// TwinCAT 3 PLC project Tc_PLCopen_OpcUa
// Title: Tc_PLCopen_OpcUa
// Company: Beckhoff Automation GmbH
// Author: Beckhoff Automation GmbH
// ProjectVersion: 2.0
// ProgramVersion: 3.1.4020.1
// libraries:
//   Tc2_Standard, * (Beckhoff Automation GmbH)
//   Tc2_System, * (Beckhoff Automation GmbH)
//   Tc2_Utilities, * (Beckhoff Automation GmbH)
//   Tc3_Module, * (Beckhoff Automation GmbH)
//   Tc3_PLCopen_OpcUa, * (Beckhoff Automation GmbH)
// project tree:
//   DUTs/ ST_ADSReadRes.TcDUT, ST_ADSReadWriteRes.TcDUT, ST_ReadListData.TcDUT, ST_ReadListDataArrayInt.TcDUT, TcSymbolInfo.TcDUT
//   GVLs/ GVL_Tests.TcGVL
//   BECKHOFF SPECIFIC helper library/DUTs/Database/ ST_UASQLState.TcDUT
//   BECKHOFF SPECIFIC helper library/DUTs/_Internal/Database/ ST_UAMethodCall_DBRecordInsertRes.TcDUT
//   BECKHOFF SPECIFIC helper library/DUTs/_Internal/MethodCall/ ST_ADSReadState.TcDUT, ST_DeviceInfo.TcDUT, ST_UAMethodCall_AdsReadDeviceInfoRes.TcDUT, ST_UAMethodCall_AdsReadStateRes.TcDUT
//   BECKHOFF SPECIFIC helper library/POUs/Database/ UA_MethodCall_DBRecordInsert.TcPOU
//   BECKHOFF SPECIFIC helper library/POUs/MethodCall/ UA_MethodCall_ADSReadDeviceInfoReq.TcPOU, UA_MethodCall_ADSReadReq.TcPOU, UA_MethodCall_ADSReadStateReq.TcPOU, UA_MethodCall_ADSReadWriteReq.TcPOU, UA_MethodCall_ADSWriteControlReq.TcPOU, UA_MethodCall_ADSWriteReq.TcPOU
//   POUs/ PRG_READ_List.TcPOU, PRG_READ_List_woConnectIdent.TcPOU, PRG_READ_List_ArrayInt.TcPOU, MAIN.TcPOU, PRG_ADSReadDeviceInfoReq.TcPOU, PRG_ADSReadReq.TcPOU, PRG_ADSWriteReq.TcPOU, PRG_ADSWriteControlReq.TcPOU, PRG_ADSReadWriteReq.TcPOU, PRG_ADSReadStateReq.TcPOU, PRG_READ.TcPOU, PRG_WRITE.TcPOU
//   Tests_Henning/DUTs/ U_Arrays2DimInOne.TcDUT, U_Arrays3DimInOne.TcDUT, ST_UAMethodCall_CallInOut1DimParam.TcDUT, ST_UAMethodCall_CallInOut1DimStringParam.TcDUT, ST_UAMethodCall_CallInOutParam.TcDUT, U_ArraysInOne.TcDUT, U_ScalarsInOne.TcDUT
//   Tests_Henning/GVLs/ GVL_ArrayTests2DimPLC.TcGVL, GVL_ArrayTests3DimPLC.TcGVL, GVL_ArrayTests.TcGVL, GVL_ScalarTests.TcGVL
//   Tests_Henning/POUs/ PRG_2DArrayTest.TcPOU, PRG_2DArrayTest_Read.TcPOU, PRG_2DArrayTest_ReadWritten.TcPOU, PRG_2DArrayTest_Write.TcPOU, PRG_3DArrayTest.TcPOU, PRG_3DArrayTest_Read.TcPOU, PRG_3DArrayTest_ReadWritten.TcPOU, PRG_3DArrayTest_Write.TcPOU, PRG_Connect_Encrypted.TcPOU, PRG_GetBrokenHandle.TcPOU, PRG_READ_List_Henning.TcPOU, PRG_ArrayTest.TcPOU, PRG_ArrayTest_Read.TcPOU, PRG_ArrayTest_ReadWritten.TcPOU, PRG_ArrayTest_Write.TcPOU, PRG_CallInOut1DimParam.TcPOU, PRG_CallInOut1DimStringParam.TcPOU, PRG_CallInOutMultiParam.TcPOU, PRG_ScalarTest.TcPOU, PRG_ScalarTest_Read.TcPOU, PRG_ScalarTest_ReadWritten.TcPOU, PRG_ScalarTest_Write.TcPOU
//   Test_CloudSample/DUTs/ ST_CloudSampleRes.TcDUT, ST_DBSQLError.TcDUT, ST_internalSQLError.TcDUT
//   Test_CloudSample/GVLs/ GVL_CloudSample.TcGVL
//   Test_CloudSample/POUs/ADS/ FB_CloudAdsSqlInsert.TcPOU
//   Test_CloudSample/POUs/ CloudSample.TcPOU, CloudSample_SQL.TcPOU
//   Test_CloudSample/POUs/Helper/ FB_BuildSQLInsert.TcPOU
//   / PlcTask.TcTTO
//   Test_Manz/DUTs/ ST_UAMethodCall_CallTestMethodArray.TcDUT, ST_UAMethodCall_CallTestMethodIntArray3Dim.TcDUT
//   Test_Manz/POUs/ PRG_CallTestMethodIntArray3Dim.TcPOU, PRG_CallTestMethodStringArray2Dim.TcPOU
// real-time tasks:
//   TASK PlcTask: cycle T#10ms, priority 20, ADS port 350

CONFIGURATION Tc_PLCopen_OpcUa
    RESOURCE PLC ON TwinCAT3
        TASK PlcTask(INTERVAL := T#10ms, PRIORITY := 20);
        PROGRAM MAIN WITH PlcTask : MAIN;
    END_RESOURCE
END_CONFIGURATION

// ---- DUTs/ST_ADSReadRes.TcDUT
TYPE ST_ADSReadRes :
STRUCT
	nNumberOfOutputArguments	: UDINT;
	nReserved					: ARRAY [1..4] OF BYTE; // padding
	stOutputArgInfo				: ST_UAMethodArgInfo;
	nReadData					: INT; 
END_STRUCT
END_TYPE

// ---- DUTs/ST_ADSReadWriteRes.TcDUT
TYPE ST_ADSReadWriteRes :
STRUCT
	nNumberOfOutputArguments	: UDINT;
	nReserved					: ARRAY [1..4] OF BYTE; // padding
	stOutputArgInfo				: ST_UAMethodArgInfo;
	arrAddr						: T_IPv4AddrArr	:=[ 0, 0, 0, 0];
END_STRUCT
END_TYPE

// ---- DUTs/ST_ReadListData.TcDUT
{attribute 'pack_mode' := '1'}
TYPE ST_ReadListData :
STRUCT
	stReadListReturnInfo	: ARRAY [1..gNodeIDCount] OF ST_UAReadListReturnInfo; // must be less than nMaxNodeIDsInList, nMaxNodeIDsInList = 10
	nIntVar1				: INT; 
	nIntVar2				: INT; 
	nIntVar3				: INT;
	nIntVar4				: INT;
	nIntVar5				: INT;
	nIntVar6				: INT;
	nIntVar7				: INT;
	nIntVar8				: INT;
	nIntVar9				: INT;
	nIntVar10				: INT;
END_STRUCT
END_TYPE

// ---- DUTs/ST_ReadListDataArrayInt.TcDUT
{attribute 'pack_mode' := '1'}
TYPE ST_ReadListDataArrayInt :
STRUCT
	stReadListReturnInfo	: ARRAY [1..gNodeIDCount_Array] OF ST_UAReadListReturnInfo; // must be less than nMaxNodeIDsInList, nMaxNodeIDsInList = 10
	nArrIntVar1				: ARRAY [1..10] OF INT; 
	nArrDintVar2			: ARRAY [1..2] OF DINT; 	
END_STRUCT
END_TYPE

// ---- DUTs/TcSymbolInfo.TcDUT
TYPE TcSymbolInfo :
STRUCT
	nAddress	: UDINT; 
	nLength		: UDINT; 
END_STRUCT
END_TYPE

// ---- BECKHOFF SPECIFIC helper library/DUTs/Database/ST_UASQLState.TcDUT
TYPE ST_UASQLState :
STRUCT
	sSQLState 		: STRING(5);
	nReserved		: ARRAY [1..2] OF BYTE; //padding
	nSQLErrorCode 	: DINT;
	nReturnCode		: UDINT;
END_STRUCT
END_TYPE

// ---- BECKHOFF SPECIFIC helper library/DUTs/_Internal/Database/ST_UAMethodCall_DBRecordInsertRes.TcDUT
TYPE ST_UAMethodCall_DBRecordInsertRes :
STRUCT
	nNumberOfOutputArguments	: UDINT;
	nReserved					: ARRAY [1..4] OF BYTE; // padding
	stOutputArgInfo				: ARRAY [1..1] OF ST_UAMethodArgInfo;
	stSQLStateInternal			: ST_UASQLState; 
END_STRUCT
END_TYPE

// ---- BECKHOFF SPECIFIC helper library/DUTs/_Internal/MethodCall/ST_ADSReadState.TcDUT
TYPE ST_ADSReadState :
STRUCT
	nAdsState			: DINT;			(* ADS state *)
	nDeviceState		: DINT;			(* Device state *)
END_STRUCT
END_TYPE

// ---- BECKHOFF SPECIFIC helper library/DUTs/_Internal/MethodCall/ST_DeviceInfo.TcDUT
TYPE ST_DeviceInfo :
STRUCT
	sDeviceName		: STRING(19);		(* ADS state *)
	nVersion		: SINT;				(* Device state *)
	nRevision		: SINT;
	nBuild			: INT;
END_STRUCT
END_TYPE

// ---- BECKHOFF SPECIFIC helper library/DUTs/_Internal/MethodCall/ST_UAMethodCall_AdsReadDeviceInfoRes.TcDUT
TYPE ST_UAMethodCall_AdsReadDeviceInfoRes :
STRUCT
	nNumberOfOutputArguments	: UDINT;
	nReserved					: ARRAY [1..4] OF BYTE; // padding
	stOutputArgInfo				: ARRAY [1..4] OF ST_UAMethodArgInfo;
	stDeviceInfo				: ST_DeviceInfo;
END_STRUCT
END_TYPE

// ---- BECKHOFF SPECIFIC helper library/DUTs/_Internal/MethodCall/ST_UAMethodCall_AdsReadStateRes.TcDUT
TYPE ST_UAMethodCall_AdsReadStateRes :
STRUCT
	nNumberOfOutputArguments	: UDINT;
	nReserved					: ARRAY [1..4] OF BYTE; // padding
	stOutputArgInfo				: ARRAY [1..3] OF ST_UAMethodArgInfo;
	stADSReadState				: ST_ADSReadState;
END_STRUCT
END_TYPE

// ---- Tests_Henning/DUTs/U_Arrays2DimInOne.TcDUT
TYPE U_Arrays2DimInOne :

UNION
	nData	: ARRAY[1..nMaxReadDataArray_2Dim] OF BYTE;
	bBool	: ARRAY[1..nArrayTestLength_2DimX, 1..nArrayTestLength_2DimY] OF BOOL;
	bByte	: ARRAY[1..nArrayTestLength_2DimX, 1..nArrayTestLength_2DimY] OF BYTE;
	nInt	: ARRAY[1..nArrayTestLength_2DimX, 1..nArrayTestLength_2DimY] OF INT;
	nUdint	: ARRAY[1..nArrayTestLength_2DimX, 1..nArrayTestLength_2DimY] OF UDINT;
	nReal	: ARRAY[1..nArrayTestLength_2DimX, 1..nArrayTestLength_2DimY] OF REAL;
	nLReal	: ARRAY[1..nArrayTestLength_2DimX, 1..nArrayTestLength_2DimY] OF LREAL;
	sString	: ARRAY[1..nArrayTestLength_2DimX, 1..nArrayTestLength_2DimY] OF STRING(80);
	wLword	: ARRAY[1..nArrayTestLength_2DimX, 1..nArrayTestLength_2DimY] OF LWORD;
	dDate	: ARRAY[1..nArrayTestLength_2DimX, 1..nArrayTestLength_2DimY] OF DT;
END_UNION

END_TYPE

// ---- Tests_Henning/DUTs/U_Arrays3DimInOne.TcDUT
TYPE U_Arrays3DimInOne :

UNION
	nData	: ARRAY[1..nMaxReadDataArray_3Dim] OF BYTE;
	bBool	: ARRAY[1..nArrayTestLength_3DimX, 1..nArrayTestLength_3DimY, 1..nArrayTestLength_3DimZ] OF BOOL;
	bByte	: ARRAY[1..nArrayTestLength_3DimX, 1..nArrayTestLength_3DimY, 1..nArrayTestLength_3DimZ] OF BYTE;
	nInt	: ARRAY[1..nArrayTestLength_3DimX, 1..nArrayTestLength_3DimY, 1..nArrayTestLength_3DimZ] OF INT;
	nUdint	: ARRAY[1..nArrayTestLength_3DimX, 1..nArrayTestLength_3DimY, 1..nArrayTestLength_3DimZ] OF UDINT;
	nReal	: ARRAY[1..nArrayTestLength_3DimX, 1..nArrayTestLength_3DimY, 1..nArrayTestLength_3DimZ] OF REAL;
	nLReal	: ARRAY[1..nArrayTestLength_3DimX, 1..nArrayTestLength_3DimY, 1..nArrayTestLength_3DimZ] OF LREAL;
	sString	: ARRAY[1..nArrayTestLength_3DimX, 1..nArrayTestLength_3DimY, 1..nArrayTestLength_3DimZ] OF STRING(80);
	wLword	: ARRAY[1..nArrayTestLength_3DimX, 1..nArrayTestLength_3DimY, 1..nArrayTestLength_3DimZ] OF LWORD;
	dDate	: ARRAY[1..nArrayTestLength_3DimX, 1..nArrayTestLength_3DimY, 1..nArrayTestLength_3DimZ] OF DT;
END_UNION

END_TYPE

// ---- Test_CloudSample/DUTs/ST_CloudSampleRes.TcDUT
TYPE ST_CloudSampleRes :
STRUCT
	nNumberOfOutputArguments	: UDINT;
	nReserved 					: ARRAY [1..4] OF BYTE;
	stOutputArgInfo				: ARRAY [1..1] of ST_UAMethodArgInfo;
	stUASQLStateInternal		: ST_UASQLState;
END_STRUCT
END_TYPE

// ---- Test_CloudSample/DUTs/ST_DBSQLError.TcDUT
TYPE ST_DBSQLError :
STRUCT
	sSQLState : STRING(5);
	nSQLErrorCode : DINT;
END_STRUCT
END_TYPE

// ---- Test_CloudSample/DUTs/ST_internalSQLError.TcDUT
TYPE ST_internalSQLError :
STRUCT
	sSQLState : STRING(5);
	dummy : ARRAY [0..1] OF BYTE;
	nSQLErrorCode : DINT;
END_STRUCT
END_TYPE

// ---- Tests_Henning/DUTs/ST_UAMethodCall_CallInOut1DimParam.TcDUT
TYPE ST_UAMethodCall_CallInOut1DimParam :
STRUCT
	nNumberOfOutputArguments	: UDINT;
	nReserved					: ARRAY [1..4] OF BYTE; // padding
	stOutputArgInfo				: ARRAY [1..1] OF ST_UAMethodArgInfo;
	//If dynamic out params are in front of others: they need to be memcpyed afterwards.
	//OutputData					: ARRAY [1..8] OF BYTE;
	//This testmethod just returns 2 DINTs so we could directly define them here
	output1						: DINT;
	output2						: DINT;  
	output3						: DINT;  
END_STRUCT
END_TYPE

// ---- Tests_Henning/DUTs/ST_UAMethodCall_CallInOut1DimStringParam.TcDUT
TYPE ST_UAMethodCall_CallInOut1DimStringParam :
STRUCT
	nNumberOfOutputArguments	: UDINT;
	nReserved					: ARRAY [1..4] OF BYTE; // padding
	stOutputArgInfo				: ARRAY [1..1] OF ST_UAMethodArgInfo;
	//If dynamic out params are in front of others: they need to be memcpyed afterwards.
	//OutputData					: ARRAY [1..8] OF BYTE;
	//This testmethod just returns 2 DINTs so we could directly define them here
	sOutArray					: ARRAY[1..3] OF STRING;
END_STRUCT
END_TYPE

// ---- Tests_Henning/DUTs/ST_UAMethodCall_CallInOutParam.TcDUT
TYPE ST_UAMethodCall_CallInOutParam :
STRUCT
	nNumberOfOutputArguments	: UDINT := 2;
	nReserved					: ARRAY [1..4] OF BYTE; // padding
	stOutputArgInfo				: ARRAY [1..2] OF ST_UAMethodArgInfo;
	//If dynamic out params are in front of others: they need to be memcpyed afterwards.
	//OutputData					: ARRAY [1..8] OF BYTE;
	//This testmethod just returns 2 DINTs so we could directly define them here
	output1						: DINT;
	output2						: DINT;  
END_STRUCT
END_TYPE

// ---- Tests_Henning/DUTs/U_ArraysInOne.TcDUT
TYPE U_ArraysInOne :

UNION
	nData	: ARRAY[1..nMaxReadDataArray] OF BYTE;
	bBool	: ARRAY[1..nArrayTestLength] OF BOOL;
	bByte	: ARRAY[1..nArrayTestLength] OF BYTE;
	nInt	: ARRAY[1..nArrayTestLength] OF INT;
	nUdint	: ARRAY[1..nArrayTestLength] OF UDINT;
	nReal	: ARRAY[1..nArrayTestLength] OF REAL;
	nLReal	: ARRAY[1..nArrayTestLength] OF LREAL;
	sString	: ARRAY[1..nArrayTestLength] OF STRING(80);
	wLword	: ARRAY[1..nArrayTestLength] OF LWORD;
END_UNION

END_TYPE

// ---- Tests_Henning/DUTs/U_ScalarsInOne.TcDUT
TYPE U_ScalarsInOne :

UNION
	nData	: ARRAY[1..nMaxReadData] OF BYTE;
	bBool	: BOOL;
	bByte	: BYTE;
	nInt	: INT;
	nUdint	: UDINT;
	nReal	: REAL;
	nLReal	: LREAL;
	sString	: STRING(255);
	wLword	: LWORD;
END_UNION

END_TYPE

// ---- Test_Manz/DUTs/ST_UAMethodCall_CallTestMethodArray.TcDUT
TYPE ST_UAMethodCall_CallTestMethodArray :
STRUCT
	nNumberOfOutputArguments	: UDINT;	(* 4*)
	nReserved					: ARRAY [1..4] OF BYTE; // padding
	stOutputArgInfo				: ARRAY [1..2] OF ST_UAMethodArgInfo;	(* 24 + 24 *)
	//If dynamic out params are in front of others: they need to be memcpyed afterwards.
	//OutputData					: ARRAY [1..8] OF BYTE;
	//This testmethod just returns 2 DINTs so we could directly define them here
	output1						: ARRAY[1..10] OF LREAL; (* 80 *)
	output2						: ARRAY[1..10] OF STRING;  (* 810 *)
END_STRUCT
END_TYPE

// ---- Test_Manz/DUTs/ST_UAMethodCall_CallTestMethodIntArray3Dim.TcDUT
TYPE ST_UAMethodCall_CallTestMethodIntArray3Dim :
STRUCT
	nNumberOfOutputArguments	: UDINT := 1;
	nReserved					: ARRAY [1..4] OF BYTE; // padding
	stOutputArgInfo				: ARRAY [1..1] OF ST_UAMethodArgInfo;
	//If dynamic out params are in front of others: they need to be memcpyed afterwards.
	//OutputData					: ARRAY [1..8] OF BYTE;
	//This testmethod just returns 2 DINTs so we could directly define them here
	output1						: ARRAY[1..3,1..3,1..3] OF DINT;
END_STRUCT
END_TYPE

// ---- GVLs/GVL_Tests.TcGVL
VAR_GLOBAL CONSTANT
	sPujaNetID				: T_AmsNetID := '172.17.214.3.1.1'; 
//	sHenningNetID			: T_AmsNetID := '172.17.214.25.1.1';

	gNodeIDCount					: UINT := 10;
	gNodeIDCount_Array				: UINT := 2;

END_VAR

// ---- Tests_Henning/GVLs/GVL_ArrayTests2DimPLC.TcGVL
VAR_GLOBAL CONSTANT
	nEndOfNodeIDVarsArray_2Dim: UINT := 9;
	nArrayTestLength_2DimX: UDINT := 4;
	nArrayTestLength_2DimY: UDINT := 2;
	//nArrayTestLength_2DimX*nArrayTestLength_2DimY*80
	nMaxReadDataArray_2Dim: UDINT := 640; 
	//sOpcUA_URL: STRING := 'opc.tcp://henningm-nb:4840';
	sOpcUA_URL: STRING := 'opc.tcp://localhost:4842';
	sNodeIDNamespace: STRING := 'TmcPLC';
END_VAR
VAR_GLOBAL
	NodeID_Identifiers: ARRAY[0..nEndOfNodeIDVarsArray_2Dim] OF STRING := 
		['GVL_ArrayTests2DimPLC.stat_BOOL_2Dim', 
		 'GVL_ArrayTests2DimPLC.stat_BSTRARRAY_2Dim',
		 'GVL_ArrayTests2DimPLC.stat_I1_2Dim', 
		 'GVL_ArrayTests2DimPLC.stat_I2_2Dim', 
		 'GVL_ArrayTests2DimPLC.stat_I4_2Dim', 
		 'GVL_ArrayTests2DimPLC.stat_R8_2Dim', 
		 'GVL_ArrayTests2DimPLC.stat_UI1_2Dim', 
		 'GVL_ArrayTests2DimPLC.stat_UI2_2Dim', 
		 'GVL_ArrayTests2DimPLC.stat_UI4_2Dim',
		 'GVL_ArrayTests2DimPLC.stat_DATE_2Dim'
	];
	NodeID_Sizes: ARRAY[0..nEndOfNodeIDVarsArray_2Dim] OF UDINT := 
		[(1 * nArrayTestLength_2DimX * nArrayTestLength_2DimY), 
		 (81 * nArrayTestLength_2DimX * nArrayTestLength_2DimY), 
		 (1 * nArrayTestLength_2DimX * nArrayTestLength_2DimY), 
		 (2 * nArrayTestLength_2DimX * nArrayTestLength_2DimY), 
		 (4 * nArrayTestLength_2DimX * nArrayTestLength_2DimY), 
		 (8 * nArrayTestLength_2DimX * nArrayTestLength_2DimY), 
		 (1 * nArrayTestLength_2DimX * nArrayTestLength_2DimY), 
		 (2 * nArrayTestLength_2DimX * nArrayTestLength_2DimY), 
		 (4 * nArrayTestLength_2DimX * nArrayTestLength_2DimY), 
		 (4 * nArrayTestLength_2DimX * nArrayTestLength_2DimY)
	];
	NodeID_DoOrDont: ARRAY[0..nEndOfNodeIDVarsArray_2Dim] OF BOOL := 
		[TRUE, //'GVL_ArrayTests3DimPLC.stat_BOOL_3Dim', 
		 TRUE, //'GVL_ArrayTests3DimPLC.stat_BSTRARRAY_3Dim',
		 TRUE, //'GVL_ArrayTests3DimPLC.stat_I1_3Dim', 
		 TRUE, //'GVL_ArrayTests3DimPLC.stat_I2_3Dim', 
		 TRUE, //'GVL_ArrayTests3DimPLC.stat_I4_3Dim', 
		 TRUE, //'GVL_ArrayTests3DimPLC.stat_R8_3Dim', 
		 TRUE, //'GVL_ArrayTests3DimPLC.stat_UI1_3Dim', 
		 TRUE, //'GVL_ArrayTests3DimPLC.stat_UI2_3Dim',  
		 TRUE, //'GVL_ArrayTests3DimPLC.stat_UI4_3Dim', 
		 FALSE //'GVL_ArrayTests3DimPLC.stat_DATE_3Dim'
	];
	NodeID_WriteCommands: ARRAY[0..nEndOfNodeIDVarsArray_2Dim] OF U_Arrays2DimInOne := [
			(bBool := [TRUE, FALSE, TRUE, FALSE, TRUE, FALSE, TRUE, FALSE]), 
	 		(sString := ['aaa', 'bbbb', 'ccccc', 'ddddddd', 'aaa', 'bbbb', 'ccccc', 'ddddddd']), 
			(bByte := [123, 124, 125, 126, 123, 124, 125, 126]), 
			(nInt := [127, 128, 129, 130,127, 128, 129, 130]), 
			(nUdint := [131, 132, 133, 134, 131, 132, 133, 134]), 
			(nLReal := [1.23456, 1.23457, 1.23458, 1.23459, 1.23456, 1.23457, 1.23458, 1.23459]), 
			(bByte := [111, 112, 113, 114, 111, 112, 113, 114]), 
			(nInt := [115, 116, 117, 118,115, 116, 117, 118]), 
			(nUdint := [119, 120, 121, 122, 119, 120, 121, 122]), 
			(dDate := [DT#2008-9-26-0:11:12, DT#2008-9-26-0:11:13, DT#2008-9-26-0:11:14, DT#2008-9-26-0:11:15, DT#2008-9-26-0:11:12, DT#2008-9-26-0:11:13, DT#2008-9-26-0:11:14, DT#2008-9-26-0:11:15]) 
	];
	NodeID_ReadResults: ARRAY[0..nEndOfNodeIDVarsArray_2Dim] OF U_Arrays2DimInOne;
	NodeID_ReadWrittenResults: ARRAY[0..nEndOfNodeIDVarsArray_2Dim] OF U_Arrays2DimInOne;
	NodeID_CheckReadWrite: ARRAY[0..nEndOfNodeIDVarsArray_2Dim] OF BOOL;
	
	//Data fields
	stat_BOOL_2Dim: 		ARRAY[1..nArrayTestLength_2DimX, 1..nArrayTestLength_2DimY] OF BOOL 	:= [TRUE, TRUE, TRUE, TRUE, FALSE, FALSE, FALSE, FALSE]; 						(*~ (OPC : 1 : enabled for OPC) *)
	stat_BSTRARRAY_2Dim: 	ARRAY[1..nArrayTestLength_2DimX, 1..nArrayTestLength_2DimY] OF STRING 	:= ['these', 'are', 'init', 'values', 'which', 'will', 'be', 'overwritten'];	(*~ (OPC : 1 : enabled for OPC) *)
	stat_I1_2Dim: 			ARRAY[1..nArrayTestLength_2DimX, 1..nArrayTestLength_2DimY] OF BYTE		:= [1, 1, 1, 1, 1, 1, 1, 1];													(*~ (OPC : 1 : enabled for OPC) *)
	stat_I2_2Dim: 			ARRAY[1..nArrayTestLength_2DimX, 1..nArrayTestLength_2DimY] OF INT		:= [1, 1, 1, 1, 1, 1, 1, 1];													(*~ (OPC : 1 : enabled for OPC) *)
	stat_I4_2Dim:			ARRAY[1..nArrayTestLength_2DimX, 1..nArrayTestLength_2DimY] OF DINT 	:= [1, 1, 1, 1, 1, 1, 1, 1];													(*~ (OPC : 1 : enabled for OPC) *)
	stat_R8_2Dim: 			ARRAY[1..nArrayTestLength_2DimX, 1..nArrayTestLength_2DimY] OF LREAL	:= [1.1, 1.1, 1.1, 1.1, 1.1, 1.1, 1.1, 1.1];									(*~ (OPC : 1 : enabled for OPC) *)
	stat_UI1_2Dim:			ARRAY[1..nArrayTestLength_2DimX, 1..nArrayTestLength_2DimY] OF BYTE		:= [1, 1, 1, 1, 1, 1, 1, 1];													(*~ (OPC : 1 : enabled for OPC) *)
	stat_UI2_2Dim: 			ARRAY[1..nArrayTestLength_2DimX, 1..nArrayTestLength_2DimY] OF UINT		:= [1, 1, 1, 1, 1, 1, 1, 1];													(*~ (OPC : 1 : enabled for OPC) *)
	stat_UI4_2Dim: 			ARRAY[1..nArrayTestLength_2DimX, 1..nArrayTestLength_2DimY] OF UDINT	:= [1, 1, 1, 1, 1, 1, 1, 1];													(*~ (OPC : 1 : enabled for OPC) *)
	stat_DATE_2Dim:			ARRAY[1..nArrayTestLength_2DimX, 1..nArrayTestLength_2DimY] OF DT		:= [DT#2014-2-20-0:11:12, DT#2014-2-20-0:11:12, DT#2014-2-20-0:11:12, DT#2014-2-20-0:11:12, DT#2014-2-20-0:11:12, DT#2014-2-20-0:11:12, DT#2014-2-20-0:11:12, DT#2014-2-20-0:11:12];													(*~ (OPC : 1 : enabled for OPC) *)
		
END_VAR

// ---- Tests_Henning/GVLs/GVL_ArrayTests3DimPLC.TcGVL
VAR_GLOBAL CONSTANT
	nEndOfNodeIDVarsArray_3Dim: UINT := 9 ;
	nArrayTestLength_3DimX: UDINT := 4;
	nArrayTestLength_3DimY: UDINT := 2;
	nArrayTestLength_3DimZ: UDINT := 2;
	//nArrayTestLength_3DimX*nArrayTestLength_3DimY*nArrayTestLength_3DimZ*80
	nMaxReadDataArray_3Dim: UDINT := 1280; 
	//sOpcUA_URL: STRING := 'opc.tcp://henningm-nb:4840';
	sOpcUA_URL: STRING := 'opc.tcp://localhost:4842';
	sNodeIDNamespace: STRING := 'TmcPLC';
END_VAR
VAR_GLOBAL
	NodeID_Identifiers: ARRAY[0..nEndOfNodeIDVarsArray_3Dim] OF STRING := 
		['GVL_ArrayTests3DimPLC.stat_BOOL_3Dim', 
		 'GVL_ArrayTests3DimPLC.stat_BSTRARRAY_3Dim',
		 'GVL_ArrayTests3DimPLC.stat_I1_3Dim', 
		 'GVL_ArrayTests3DimPLC.stat_I2_3Dim', 
		 'GVL_ArrayTests3DimPLC.stat_I4_3Dim', 
		 'GVL_ArrayTests3DimPLC.stat_R8_3Dim', 
		 'GVL_ArrayTests3DimPLC.stat_UI1_3Dim', 
		 'GVL_ArrayTests3DimPLC.stat_UI2_3Dim',  
		 'GVL_ArrayTests3DimPLC.stat_UI4_3Dim', 
		 'GVL_ArrayTests3DimPLC.stat_DATE_3Dim'
	];
	NodeID_Sizes: ARRAY[0..nEndOfNodeIDVarsArray_3Dim] OF UDINT := 
		[(1 * nArrayTestLength_3DimX * nArrayTestLength_3DimY * nArrayTestLength_3DimZ), 
		 (81 * nArrayTestLength_3DimX * nArrayTestLength_3DimY * nArrayTestLength_3DimZ), 
		 (1 * nArrayTestLength_3DimX * nArrayTestLength_3DimY * nArrayTestLength_3DimZ), 
		 (2 * nArrayTestLength_3DimX * nArrayTestLength_3DimY * nArrayTestLength_3DimZ), 
		 (4 * nArrayTestLength_3DimX * nArrayTestLength_3DimY  * nArrayTestLength_3DimZ), 
		 (8 * nArrayTestLength_3DimX * nArrayTestLength_3DimY  * nArrayTestLength_3DimZ), 
		 (1 * nArrayTestLength_3DimX * nArrayTestLength_3DimY  * nArrayTestLength_3DimZ), 
		 (2 * nArrayTestLength_3DimX * nArrayTestLength_3DimY  * nArrayTestLength_3DimZ), 
	     (4 * nArrayTestLength_3DimX * nArrayTestLength_3DimY  * nArrayTestLength_3DimZ), 
	     (4 * nArrayTestLength_3DimX * nArrayTestLength_3DimY  * nArrayTestLength_3DimZ)
	];
	NodeID_DoOrDont: ARRAY[0..nEndOfNodeIDVarsArray_3Dim] OF BOOL := 
		[TRUE, //'GVL_ArrayTests3DimPLC.stat_BOOL_3Dim', 
		 TRUE, //'GVL_ArrayTests3DimPLC.stat_BSTRARRAY_3Dim',
		 TRUE, //'GVL_ArrayTests3DimPLC.stat_I1_3Dim', 
		 TRUE, //'GVL_ArrayTests3DimPLC.stat_I2_3Dim', 
		 TRUE, //'GVL_ArrayTests3DimPLC.stat_I4_3Dim', 
		 TRUE, //'GVL_ArrayTests3DimPLC.stat_R8_3Dim', 
		 TRUE, //'GVL_ArrayTests3DimPLC.stat_UI1_3Dim', 
		 TRUE, //'GVL_ArrayTests3DimPLC.stat_UI2_3Dim',  
		 TRUE, //'GVL_ArrayTests3DimPLC.stat_UI4_3Dim', 
		 FALSE //'GVL_ArrayTests3DimPLC.stat_DATE_3Dim'
	];
	NodeID_WriteCommands: ARRAY[0..nEndOfNodeIDVarsArray_3Dim] OF U_Arrays3DimInOne := [
			(bBool := [TRUE, FALSE, TRUE, FALSE, TRUE, FALSE, TRUE, FALSE, TRUE, FALSE, TRUE, FALSE, TRUE, FALSE, TRUE, FALSE]), 
	 		(sString := ['aaa', 'bbbb', 'ccccc', 'ddddddd', 'aaa', 'bbbb', 'ccccc', 'ddddddd', 'aaa', 'bbbb', 'ccccc', 'ddddddd', 'aaa', 'bbbb', 'ccccc', 'ddddddd']), 
			(bByte := [123, 124, 125, 126, 123, 124, 125, 126, 123, 124, 125, 126, 123, 124, 125, 126]), 
			(nInt := [127, 128, 129, 130,127, 128, 129, 130, 127, 128, 129, 130,127, 128, 129, 130]), 
			(nUdint := [131, 132, 133, 134, 131, 132, 133, 134, 131, 132, 133, 134, 131, 132, 133, 134]), 
			(nLReal := [1.23456, 1.23457, 1.23458, 1.23459, 1.23456, 1.23457, 1.23458, 1.23459, 1.23456, 1.23457, 1.23458, 1.23459, 1.23456, 1.23457, 1.23458, 1.23459]), 
			(bByte := [111, 112, 113, 114, 111, 112, 113, 114, 111, 112, 113, 114, 111, 112, 113, 114]), 
			(nInt := [115, 116, 117, 118,115, 116, 117, 118, 115, 116, 117, 118,115, 116, 117, 118]), 
			(nUdint := [119, 120, 121, 122, 119, 120, 121, 122, 119, 120, 121, 122, 119, 120, 121, 122]), 
			(dDate := [DT#2008-9-26-0:11:12, DT#2008-9-26-0:11:13, DT#2008-9-26-0:11:14, DT#2008-9-26-0:11:15, DT#2008-9-26-0:11:12, DT#2008-9-26-0:11:13, DT#2008-9-26-0:11:14, DT#2008-9-26-0:11:15, DT#2008-9-26-0:11:12, DT#2008-9-26-0:11:13, DT#2008-9-26-0:11:14, DT#2008-9-26-0:11:15, DT#2008-9-26-0:11:12, DT#2008-9-26-0:11:13, DT#2008-9-26-0:11:14, DT#2008-9-26-0:11:15]) 
	];
	NodeID_ReadResults: ARRAY[0..nEndOfNodeIDVarsArray_3Dim] OF U_Arrays3DimInOne;
	NodeID_ReadWrittenResults: ARRAY[0..nEndOfNodeIDVarsArray_3Dim] OF U_Arrays3DimInOne;
	NodeID_CheckReadWrite: ARRAY[0..nEndOfNodeIDVarsArray_3Dim] OF BOOL;
	
	//Data fields
	test : BOOL; (*~ (OPC : 1 : enabled for OPC) *)
	stat_BOOL_3Dim: 		ARRAY[1..nArrayTestLength_3DimX, 1..nArrayTestLength_3DimY, 1..nArrayTestLength_3DimZ] OF BOOL 	:= [TRUE, TRUE, TRUE, TRUE, FALSE, FALSE, FALSE, FALSE,TRUE, TRUE, TRUE, TRUE, FALSE, FALSE, FALSE, FALSE]; 						(*~ (OPC : 1 : enabled for OPC) *)
	stat_BSTRARRAY_3Dim: 	ARRAY[1..nArrayTestLength_3DimX, 1..nArrayTestLength_3DimY, 1..nArrayTestLength_3DimZ] OF STRING 	:= ['these', 'are', 'init', 'values', 'which', 'will', 'be', 'overwritten', 'these', 'are', 'init', 'values', 'which', 'will', 'be', 'overwritten'];	(*~ (OPC : 1 : enabled for OPC) *)
	stat_I1_3Dim: 			ARRAY[1..nArrayTestLength_3DimX, 1..nArrayTestLength_3DimY, 1..nArrayTestLength_3DimZ] OF BYTE		:= [1, 1, 1, 1, 1, 1, 1, 1, 1, 1, 1, 1, 1, 1, 1, 1];													(*~ (OPC : 1 : enabled for OPC) *)
	stat_I2_3Dim: 			ARRAY[1..nArrayTestLength_3DimX, 1..nArrayTestLength_3DimY, 1..nArrayTestLength_3DimZ] OF INT		:= [1, 1, 1, 1, 1, 1, 1, 1, 1, 1, 1, 1, 1, 1, 1, 1];													(*~ (OPC : 1 : enabled for OPC) *)
	stat_I4_3Dim:			ARRAY[1..nArrayTestLength_3DimX, 1..nArrayTestLength_3DimY, 1..nArrayTestLength_3DimZ] OF DINT 	:= [1, 1, 1, 1, 1, 1, 1, 1, 1, 1, 1, 1, 1, 1, 1, 1];													(*~ (OPC : 1 : enabled for OPC) *)
	stat_R8_3Dim: 			ARRAY[1..nArrayTestLength_3DimX, 1..nArrayTestLength_3DimY, 1..nArrayTestLength_3DimZ] OF LREAL	:= [1.1, 1.1, 1.1, 1.1, 1.1, 1.1, 1.1, 1.1, 1.1, 1.1, 1.1, 1.1, 1.1, 1.1, 1.1, 1.1];									(*~ (OPC : 1 : enabled for OPC) *)
	stat_UI1_3Dim:			ARRAY[1..nArrayTestLength_3DimX, 1..nArrayTestLength_3DimY, 1..nArrayTestLength_3DimZ] OF BYTE		:= [1, 1, 1, 1, 1, 1, 1, 1, 1, 1, 1, 1, 1, 1, 1, 1];													(*~ (OPC : 1 : enabled for OPC) *)
	stat_UI2_3Dim: 			ARRAY[1..nArrayTestLength_3DimX, 1..nArrayTestLength_3DimY, 1..nArrayTestLength_3DimZ] OF UINT		:= [1, 1, 1, 1, 1, 1, 1, 1, 1, 1, 1, 1, 1, 1, 1, 1];													(*~ (OPC : 1 : enabled for OPC) *)
	stat_UI4_3Dim: 			ARRAY[1..nArrayTestLength_3DimX, 1..nArrayTestLength_3DimY, 1..nArrayTestLength_3DimZ] OF UDINT	:= [1, 1, 1, 1, 1, 1, 1, 1,1, 1, 1, 1, 1, 1, 1, 1];													(*~ (OPC : 1 : enabled for OPC) *)
	stat_DATE_3Dim:			ARRAY[1..nArrayTestLength_3DimX, 1..nArrayTestLength_3DimY, 1..nArrayTestLength_3DimZ] OF DT	:= [DT#2014-2-20-0:11:12, DT#2014-2-20-0:11:12, DT#2014-2-20-0:11:12, DT#2014-2-20-0:11:12, DT#2014-2-20-0:11:12, DT#2014-2-20-0:11:12, DT#2014-2-20-0:11:12, DT#2014-2-20-0:11:12, DT#2014-2-20-0:11:12, DT#2014-2-20-0:11:12, DT#2014-2-20-0:11:12, DT#2014-2-20-0:11:12, DT#2014-2-20-0:11:12, DT#2014-2-20-0:11:12, DT#2014-2-20-0:11:12, DT#2014-2-20-0:11:12];													(*~ (OPC : 1 : enabled for OPC) *)
		
END_VAR

// ---- Test_CloudSample/GVLs/GVL_CloudSample.TcGVL
VAR_GLOBAL

	(* Variables for Hardware *)
	b_Light_1	AT%Q*			: BOOL;	(*~ (OPC : 1 : enabled for OPC) *)
	b_Light_2	AT%Q*			: BOOL;	(*~ (OPC : 1 : enabled for OPC) *)
	b_Light_3	AT%Q*			: BOOL;	(*~ (OPC : 1 : enabled for OPC) *)
	b_Light_4	AT%Q*			: BOOL;	(*~ (OPC : 1 : enabled for OPC) *)

	b_Button_1	AT%I*			: BOOL;	(*~ (OPC : 1 : enabled for OPC) *)
	b_Button_2	AT%I*			: BOOL;	(*~ (OPC : 1 : enabled for OPC) *)
	b_Button_3	AT%I*			: BOOL;	(*~ (OPC : 1 : enabled for OPC) *)
	b_Button_4	AT%I*			: BOOL;	(*~ (OPC : 1 : enabled for OPC) *)
	
	us_Poti_1	AT%I*			: INT;	(*~ (OPC : 1 : enabled for OPC) *)
	us_Poti_2 	AT%I*			: INT;	(*~ (OPC : 1 : enabled for OPC) *)
	us_Poti_3	AT%I*			: INT;	(*~ (OPC : 1 : enabled for OPC) *)
	us_Poti_4	AT%I*			: INT;	(*~ (OPC : 1 : enabled for OPC) *)

END_VAR

VAR_GLOBAL CONSTANT
	(*	Variables for Cloud demo *)
	MAX_DATA_ACCURACY			: INT := 4;
END_VAR

// ---- Tests_Henning/GVLs/GVL_ArrayTests.TcGVL
VAR_GLOBAL CONSTANT
	nEndOfNodeIDVarsArray: UINT := 8;
	nArrayTestLength: UDINT := 4;
	///nArrayTestLength*80
	nMaxReadDataArray: UDINT := 320;
	sOpcUA_URL: STRING := 'opc.tcp://localhost:4841';
	sNodeIDNamespace: STRING := 'PLC1';
END_VAR
VAR_GLOBAL
	NodeID_Identifiers: ARRAY[0..nEndOfNodeIDVarsArray] OF STRING := ['GVL_static.stat_BOOL', 'GVL_static.stat_BSTRARRAY', 'GVL_static.stat_I1', 'GVL_static.stat_I2', 'GVL_static.stat_I4', 'GVL_static.stat_R8', 'GVL_static.stat_UI1', 'GVL_static.stat_UI2', 'GVL_static.stat_UI4'];
	NodeID_Sizes: ARRAY[0..nEndOfNodeIDVarsArray] OF UDINT := [(1 * nArrayTestLength), (81 * nArrayTestLength), (1 * nArrayTestLength), (2 * nArrayTestLength), (4 * nArrayTestLength), (8 * nArrayTestLength), (1 * nArrayTestLength), (2 * nArrayTestLength), (4 * nArrayTestLength)];
	NodeID_WriteCommands: ARRAY[0..nEndOfNodeIDVarsArray] OF U_ArraysInOne := [(bBool := [TRUE, FALSE, TRUE, FALSE]), (sString := ['aaa', 'bbbb', 'ccccc', 'ddddddd']), (bByte := [123, 124, 125, 126]), (nInt := [127, 128, 129, 130]), (nUdint := [131, 132, 133, 134]), (nLReal := [1.23456, 1.23457, 1.23458, 1.23459]), (bByte := [111, 112, 113, 114]), (nInt := [115, 116, 117, 118]), (nUdint := [119, 120, 121, 122])];
	NodeID_ReadResults: ARRAY[0..nEndOfNodeIDVarsArray] OF U_ArraysInOne;
	NodeID_ReadWrittenResults: ARRAY[0..nEndOfNodeIDVarsArray] OF U_ArraysInOne;
	NodeID_CheckReadWrite: ARRAY[0..nEndOfNodeIDVarsArray] OF BOOL;
END_VAR

// ---- Tests_Henning/GVLs/GVL_ScalarTests.TcGVL
VAR_GLOBAL CONSTANT
	nEndOfNodeIDVars	: UINT := 8;
	nMaxReadData		: UDINT := 255;
	sOpcUA_URL			: STRING := 'opc.tcp://localhost:4841';
	sNodeIDNamespace	: STRING := 'PLC1';
END_VAR
VAR_GLOBAL
	NodeID_Identifiers		: ARRAY[0..nEndOfNodeIDVars] OF STRING := ['GVL_static.stat_BOOL1x', 'GVL_static.stat_BSTR_0', 'GVL_static.stat_I1x', 'GVL_static.stat_I2x', 'GVL_static.stat_I4x', 'GVL_static.stat_R8x', 'GVL_static.stat_UI1x', 'GVL_static.stat_UI2x', 'GVL_static.stat_UI4x'];
	NodeID_Sizes			: ARRAY[0..nEndOfNodeIDVars] OF UDINT := [1, 255, 1, 2, 4, 8, 1, 2, 4];
	NodeID_WriteCommands	: ARRAY[0..nEndOfNodeIDVars] OF U_ScalarsInOne := [(bBool := TRUE), (sString := 'WriteTest'), (bByte := 123), (nInt := 124), (nUdint := 125), (nLReal := 1.23456), (bByte := 111), (nInt := 112), (nUdint := 113)];
	NodeID_ReadResults		: ARRAY[0..nEndOfNodeIDVars] OF U_ScalarsInOne;
	NodeID_ReadWrittenResults: ARRAY[0..nEndOfNodeIDVars] OF U_ScalarsInOne;
	NodeID_CheckReadWrite	: ARRAY[0..nEndOfNodeIDVars] OF BOOL;
END_VAR

// ---- POUs/MAIN.TcPOU
PROGRAM MAIN
VAR	
	diVar1			: DINT := 22; 		(* ~ (OPC : 1 : enabled for OPC) *)
	diVar2			: DINT := 33; 		(* ~ (OPC : 1 : enabled for OPC) *)		
	iVar1			: INT := 11; 		(* ~ (OPC : 1 : enabled for OPC) *)
	iVar2			: INT := 55; 		(* ~ (OPC : 1 : enabled for OPC) *)
	
	bVar			: BOOL; 		(* ~ (OPC : 1 : enabled for OPC) *)
	nDint			: DINT;			(* ~ (OPC : 1 : enabled for OPC) *)
	iVar	 AT%MB0	: INT := 45;	(* ~ (OPC : 1 : enabled for OPC) *)
	iCount			: INT := 66;	(* ~ (OPC : 1 : enabled for OPC) *)
	sString1		: STRING(5) := 'OPCUA'; (* ~ (OPC : 1 : enabled for OPC) *)
	
	iCounter		: INT;	(*~(OPC:1:enabled)*)
	
	iArrayIntVar1	: ARRAY [1..10] OF INT := [10(22)]; 		(* ~ (OPC : 1 : enabled for OPC) *)
	diArrayDintVar2	: ARRAY [1..2] OF DINT := [2(4444)]; 		(* ~ (OPC : 1 : enabled for OPC) *)
END_VAR

iCounter := iCounter + 1; 

// ************ test programs **************
PRG_READ();
PRG_WRITE();

// ************ ADS test programs **************
PRG_ADSReadReq(); 
PRG_ADSWriteReq();
PRG_ADSReadDeviceInfoReq();
PRG_ADSReadStateReq();
PRG_ADSWriteControlReq();
PRG_ADSReadWriteReq();

//************ Read List programs
PRG_READ_List_woConnectIdent();
PRG_READ_List();
PRG_READ_List_ArrayInt();

// ************ Cloud test program **************
CloudSample_SQL();

// ************ Manz test programs **************
PRG_CallTestMethodStringArray2Dim();
PRG_CallTestMethodIntArray3Dim();

END_PROGRAM

// ---- POUs/PRG_READ.TcPOU
PROGRAM PRG_READ
VAR
	fbUA_Connect			: UA_Connect;
	SessionConnectInfo		: ST_UASessionConnectInfo;
	sOpcUA_URL				: STRING(MAX_STRING_LENGTH);
	nConnectionHdl			: DWORD;

	fbUA_GetNamespaceIndex 	: UA_GetNamespaceIndex;
	nNamespaceIndex			: UINT;

	fbUA_NodeGetHandle		: UA_NodeGetHandle;
	NodeID					: ST_UANodeID;
	nNodeHdl				: DWORD;

	fbUA_Read				: UA_Read;
	stIndexRange			: ARRAY [1..nMaxIndexRange] OF ST_UAIndexRange;
	nIndexRangeCount		: UINT;
	stNodeAddInfo			: ST_UANodeAdditionalInfo;
	nReadData				: DINT; 		// change the data type according to the variable type to be read
	bReadData				: BOOL; 
	sReadData				: STRING(4);
	cbData_R				: UDINT;
	
	fbUA_NodeReleaseHandle	: UA_NodeReleaseHandle;

	fbUA_Disconnect		: UA_Disconnect;

	iState		: INT;
	bTest		: BOOL:= TRUE;
	bDone		: BOOL;
	bBusy		: BOOL;
	bError		: BOOL;
	nErrorID	: DWORD;
END_VAR


CASE iState OF
0:	(* idle *)
	IF bTest THEN
		bTest		:= FALSE;
		bError		:= FALSE;
		nErrorID	:= 0;

		(* Parameterize *)
		sOpcUA_URL						:= 'opc.tcp://Pujak-nb:4840';	(* OpcUA Url of the device with ip address *)

		SessionConnectInfo.tConnectTimeout 		:= T#1S;
		SessionConnectInfo.tSessionTimeout 		:= T#1S;
		SessionConnectInfo.sApplicationName		:= '';
//		SessionConnectInfo.sApplicationUri 		:= '';
		SessionConnectInfo.eSecurityMode 		:= eUASecurityMsgMode_None;
		SessionConnectInfo.eSecurityPolicyUri 	:= eUASecurityPolicy_None;
		SessionConnectInfo.eTransportProfileUri := eUATransportProfileUri_UATcp;

(*		nIndexRange[1].nStartIndex := 0;
		nIndexRange[1].nEndIndex := 1;
		nIndexRange[1].bRangeAccess := TRUE; *)
		stNodeAddInfo.nIndexRangeCount := nIndexRangeCount;
		stNodeAddInfo.stIndexRange := stIndexRange;
		iState	:= iState + 1;
	END_IF

1:	(* open UA session *)
	fbUA_Connect(
		Execute				:= TRUE,
		ServerURL			:= sOpcUA_URL,
		SessionConnectInfo	:= SessionConnectInfo,
		Timeout				:= T#5S,
		ConnectionHdl		=> nConnectionHdl
	);

	IF NOT fbUA_Connect.Busy THEN
		fbUA_Connect(Execute := FALSE);

		IF NOT fbUA_Connect.Error THEN
			(* session open *)
			iState := iState + 1;
		ELSE
			bError			:= TRUE;
			nErrorID		:= fbUA_Connect.ErrorID;
			nConnectionHdl	:= 0;
			iState 			:= 0; (* idle *)
		END_IF
	END_IF


2:	(* GetNS Index *)
	fbUA_GetNamespaceIndex(
		Execute			:= TRUE,
		ConnectionHdl	:= nConnectionHdl,
		NamespaceUri	:= 'PLC2',
		NamespaceIndex	=> nNamespaceIndex
	);

	IF NOT fbUA_GetNamespaceIndex.Busy THEN
		fbUA_GetNamespaceIndex(Execute := FALSE);
		IF NOT fbUA_GetNamespaceIndex.Error THEN
			(* session closed *)
			iState 		:= iState + 1; (* idle *)
		ELSE
			bError		:= TRUE;
			nErrorID	:= fbUA_GetNamespaceIndex.ErrorID;
			iState 		:= 6; (* idle *)
		END_IF
	END_IF


3:	(* Get Node Handle *)
	NodeID.eIdentifierType := eUAIdentifierType_String;
	NodeID.nNamespaceIndex := nNamespaceIndex;
	NodeID.sIdentifier	:= 'MAIN.bVar';
	fbUA_NodeGetHandle(
		Execute			:= TRUE,
		ConnectionHdl	:= nConnectionHdl,
		NodeID			:= NodeID,
		NodeHdl			=> nNodeHdl
	);

	IF NOT fbUA_NodeGetHandle.Busy THEN
		fbUA_NodeGetHandle(Execute := FALSE);

		IF NOT fbUA_NodeGetHandle.Error THEN
			(* session closed *)
			iState 					:= iState + 1; (* idle *)
		ELSE
			bError		:= TRUE;
			nErrorID	:= fbUA_NodeGetHandle.ErrorID;
			iState 		:= 6; (* idle *)
		END_IF
	END_IF


4: 	(* UA_Read *)
	fbUA_Read(
		Execute			:= TRUE,
		ConnectionHdl	:= nConnectionHdl,
		NodeHdl			:= nNodeHdl,
		cbData			:= 4,
		stNodeAddInfo 	:= stNodeAddInfo,
		pVariable		:= ADR(bReadData)
		);

	IF NOT fbUA_Read.Busy THEN
		fbUA_Read( Execute := FALSE, cbData_R => cbData_R);

		IF NOT fbUA_Read.Error THEN
			(* session closed *)
			iState 		:= iState + 1; (* idle *)
		ELSE
			bError		:= TRUE;
			nErrorID	:= fbUA_Read.ErrorID;
			iState 		:= 6; (* idle *)
		END_IF
	END_IF


5:	(* Release Node Handle *)
	fbUA_NodeReleaseHandle(
		Execute			:= TRUE,
		ConnectionHdl	:= nConnectionHdl,
		NodeHdl			:= nNodeHdl
	);

	IF NOT fbUA_NodeReleaseHandle.Busy THEN
		fbUA_NodeReleaseHandle(Execute := FALSE);

		IF NOT fbUA_NodeReleaseHandle.Error THEN
			(* session closed *)
			iState 		:= iState + 1; (* idle *)
		ELSE
			bError		:= TRUE;
			nErrorID	:= fbUA_NodeReleaseHandle.ErrorID;
			iState 		:= 6; (* idle *)
		END_IF
	END_IF


6:	(* close session *)
	fbUA_Disconnect(
		Execute			:= TRUE,
		ConnectionHdl	:= nConnectionHdl
	);

	IF NOT fbUA_Disconnect.Busy THEN
		fbUA_Disconnect(Execute := FALSE);
		bBusy := FALSE;
		IF NOT fbUA_Disconnect.Error THEN
			(* session closed *)
			iState 		:= 0; (* idle *)
			IF NOT bError THEN 
				bDone 	:= TRUE;
			END_IF
		ELSE
			bError			:= TRUE;
			nErrorID		:= fbUA_Disconnect.ErrorID;
			iState 			:= 0; (* idle *)
			nConnectionHdl	:= 0;
		END_IF
	END_IF
END_CASE

END_PROGRAM

// ---- POUs/PRG_WRITE.TcPOU
PROGRAM PRG_WRITE
VAR
	fbUA_Connect			: UA_Connect;
	SessionConnectInfo		: ST_UASessionConnectInfo;
	sOpcUA_URL				: STRING(MAX_STRING_LENGTH);
	nConnectionHdl			: DWORD;

	fbUA_GetNamespaceIndex 	: UA_GetNamespaceIndex;
	nNamespaceIndex			: UINT;

	fbUA_NodeGetHandle		: UA_NodeGetHandle;
	NodeID					: ST_UANodeID;
	nNodeHdl				: DWORD;

	fbUA_Write				: UA_Write;
	stIndexRange			: ARRAY [1..nMaxIndexRange] OF ST_UAIndexRange;
	nIndexRangeCount		: UINT;
	stNodeAddInfo			: ST_UANodeAdditionalInfo;
	nWriteData				: DINT := 45;		// change according to the type of variable
	cbData					: UDINT;
	
	fbUA_NodeReleaseHandle	: UA_NodeReleaseHandle;

	fbUA_Disconnect			: UA_Disconnect;

	iState			: INT;
	bTest			: BOOL := TRUE;
	bDone			: BOOL;
	bBusy			: BOOL;
	bError			: BOOL;
	nErrorID		: DWORD;
END_VAR

CASE iState OF
0:	(* idle *)
	IF bTest THEN
		bTest	:= FALSE;
		bError	:= FALSE;
		nErrorID	:= 0;

		(* Parameterize *)
		sOpcUA_URL						:= 'opc.tcp://Pujak-nb:4840';	(* OpcUA Url of the device with ip address *)

		SessionConnectInfo.tConnectTimeout 		:= T#1S;
		SessionConnectInfo.tSessionTimeout 		:= T#1S;
		SessionConnectInfo.sApplicationName		:= '';
//		SessionConnectInfo.sApplicationUri 		:= '';
		SessionConnectInfo.eSecurityMode 		:= eUASecurityMsgMode_None;
		SessionConnectInfo.eSecurityPolicyUri 	:= eUASecurityPolicy_None;
		SessionConnectInfo.eTransportProfileUri := eUATransportProfileUri_UATcp;

		stNodeAddInfo.nIndexRangeCount := nIndexRangeCount;
		stNodeAddInfo.stIndexRange := stIndexRange;
		iState	:= iState + 1;
	END_IF

1:	(* open UA session *)
	fbUA_Connect(
		Execute				:= TRUE,
		ServerURL			:= sOpcUA_URL,
		SessionConnectInfo	:= SessionConnectInfo,
		Timeout				:= T#5S,
		ConnectionHdl		=> nConnectionHdl
	);

	IF NOT fbUA_Connect.Busy THEN
		fbUA_Connect(Execute := FALSE);

		IF NOT fbUA_Connect.Error THEN
			(* session open *)
			iState := iState + 1;
		ELSE
			bError			:= TRUE;
			nErrorID		:= fbUA_Connect.ErrorID;
			nConnectionHdl	:= 0;
			iState 			:= 0; (* idle *)
		END_IF
	END_IF


2:	(* GetNS Index *)
	fbUA_GetNamespaceIndex(
		Execute			:= TRUE,
		ConnectionHdl	:= nConnectionHdl,
		NamespaceUri	:= 'PLC2',
		NamespaceIndex	=> nNamespaceIndex
	);

	IF NOT fbUA_GetNamespaceIndex.Busy THEN
		fbUA_GetNamespaceIndex(Execute := FALSE);

		IF NOT fbUA_GetNamespaceIndex.Error THEN
			(* session closed *)
			iState 		:= iState + 1; (* idle *)
		ELSE
			bError		:= TRUE;
			nErrorID	:= fbUA_GetNamespaceIndex.ErrorID;
			iState 		:= 6; (* idle *)
		END_IF
	END_IF


3:	(* Get Node Handle *)
	NodeID.eIdentifierType := eUAIdentifierType_String;
	NodeID.nNamespaceIndex := nNamespaceIndex;
	NodeID.sIdentifier	:= 'MAIN.nDint';
	fbUA_NodeGetHandle(
		Execute			:= TRUE,
		ConnectionHdl	:= nConnectionHdl,
		NodeID			:= NodeID,
		NodeHdl			=> nNodeHdl
	);

	IF NOT fbUA_NodeGetHandle.Busy THEN
		fbUA_NodeGetHandle(Execute := FALSE);

		IF NOT fbUA_NodeGetHandle.Error THEN
			(* session closed *)
			iState 		:= iState + 1; (* idle *)
		ELSE
			bError		:= TRUE;
			nErrorID	:= fbUA_NodeGetHandle.ErrorID;
			iState 		:= 6; (* idle *)
		END_IF
	END_IF


4: 	(* UA_Write *)
	fbUA_Write(
		Execute			:= TRUE,
		ConnectionHdl	:= nConnectionHdl,
		NodeHdl			:= nNodeHdl,
		stNodeAddInfo	:= stNodeAddInfo,
		cbData			:= SIZEOF(nWriteData),
		pVariable		:= ADR(nWriteData)
		);

	IF NOT fbUA_Write.Busy THEN
		fbUA_Write(
			Execute 	:= FALSE,
			pVariable	:= ADR(nWriteData));

		IF NOT fbUA_Write.Error THEN
			(* session closed *)
			iState 		:= iState + 1; (* idle *)
		ELSE
			bError		:= TRUE;
			nErrorID	:= fbUA_Write.ErrorID;
			iState 		:= 6; (* idle *)
		END_IF
	END_IF


5:	(* Release Node Handle *)
	fbUA_NodeReleaseHandle(
		Execute			:= TRUE,
		ConnectionHdl	:= nConnectionHdl,
		NodeHdl			:= nNodeHdl
	);

	IF NOT fbUA_NodeReleaseHandle.Busy THEN
		fbUA_NodeReleaseHandle(Execute := FALSE);

		IF NOT fbUA_NodeReleaseHandle.Error THEN
			(* session closed *)
			iState 		:= iState + 1; (* idle *)
		ELSE
			bError		:= TRUE;
			nErrorID	:= fbUA_NodeReleaseHandle.ErrorID;
			iState 		:= 6; (* idle *)
		END_IF
	END_IF


6:	(* close session *)
	fbUA_Disconnect(
		Execute			:= TRUE,
		ConnectionHdl	:= nConnectionHdl
	);

	IF NOT fbUA_Disconnect.Busy THEN
		fbUA_Disconnect(Execute := FALSE);
		bBusy := FALSE; 
		IF NOT fbUA_Disconnect.Error THEN
			(* session closed *)
			iState 		:= 0; (* idle *)
			IF NOT bError THEN 
				bDone 	:= TRUE;
			END_IF
		ELSE
			bError			:= TRUE;
			nErrorID		:= fbUA_Disconnect.ErrorID;
			iState 			:= 0; (* idle *)
			nConnectionHdl	:= 0;
		END_IF
	END_IF
END_CASE

END_PROGRAM

// ---- POUs/PRG_ADSReadReq.TcPOU
PROGRAM PRG_ADSReadReq
VAR
	fbUA_Connect			: UA_Connect;
	SessionConnectInfo		: ST_UASessionConnectInfo;
	sOpcUA_URL				: STRING(MAX_STRING_LENGTH);
	nConnectionHdl			: DWORD;

	fbUA_GetNamespaceIndex 	: UA_GetNamespaceIndex;
	nNamespaceIndex			: UINT;
	
	fbUA_MethodCall_ADSReadReq	: UA_MethodCall_ADSReadReq;
	stADSReadRes				: ST_ADSReadRes;	// the Read variable is inside this struct
	
	stOutputArgInfo				: ARRAY [1..nNumberOfOutputArguments] OF ST_UAMethodArgInfo;
	
	fbUA_NodeReleaseHandle		: UA_NodeReleaseHandle;
	
	fbUA_Disconnect				: UA_Disconnect;
		
	bTest		: BOOL:= TRUE;
	bDone		: BOOL;
	bBusy		: BOOL;
	bError		: BOOL;
	nErrorID	: DWORD;
	iState		: INT;	
END_VAR
VAR CONSTANT
	nNumberOfOutputArguments	: UDINT := 1;
END_VAR


CASE iState OF
0:	(* idle *)
	IF bTest THEN
		bTest		:= FALSE;
		bError		:= FALSE;
		nErrorID	:= 0;

		(* Parameterize *)
		sOpcUA_URL						:= 'opc.tcp://localhost:4840';	(* OpcUA Url of the device with ip address *)

		SessionConnectInfo.tConnectTimeout 	:= t#1s;
		SessionConnectInfo.tSessionTimeout 	:= t#1s;
		SessionConnectInfo.sApplicationName	:= '';
//		SessionConnectInfo.sApplicationUri 	:= '';
		SessionConnectInfo.eSecurityMode 		:= eUASecurityMsgMode_None;
		SessionConnectInfo.eSecurityPolicyUri 	:= eUASecurityPolicy_None;
		SessionConnectInfo.eTransportProfileUri := eUATransportProfileUri_UATcp;

		iState	:= iState + 1;	(* open ua session *)
	END_IF

1:	(* open UA session *)
	fbUA_Connect(
		Execute				:= TRUE,
		ServerURL			:= sOpcUA_URL,
		SessionConnectInfo	:= SessionConnectInfo,
		Timeout				:= T#5S,
		ConnectionHdl		=> nConnectionHdl
	);

	IF NOT fbUA_Connect.Busy THEN
		fbUA_Connect(Execute := FALSE);

		IF NOT fbUA_Connect.Error THEN
			(* session open *)
			iState := iState + 1;	(* get namespace index *)
		ELSE
			bError			:= TRUE;
			nErrorID		:= fbUA_Connect.ErrorID;
			nConnectionHdl	:= 0;
			iState 			:= 0; (* idle *)
		END_IF
	END_IF


2:	(* GetNS Index *)
	fbUA_GetNamespaceIndex(
		Execute			:= TRUE,
		ConnectionHdl	:= nConnectionHdl,
		NamespaceUri	:= 'ADSAMS',
		NamespaceIndex	=> nNamespaceIndex
	);

	IF NOT fbUA_GetNamespaceIndex.Busy THEN
		fbUA_GetNamespaceIndex(Execute := FALSE);

		IF NOT fbUA_GetNamespaceIndex.Error THEN
			(* session closed *)
			iState 		:= iState + 1; (* method *)
		ELSE
			bError		:= TRUE;
			nErrorID	:= fbUA_GetNamespaceIndex.ErrorID;
			iState 		:= 4; (* close session *)
		END_IF
	END_IF

3:	(*  Method  *)
	stOutputArgInfo[1].nLenData := SIZEOF(stADSReadRes.nReadData); 
	fbUA_MethodCall_ADSReadReq(
		bExecute		:= TRUE,
		nConnectionHdl	:= nConnectionHdl,
		nNamespaceIndex	:= nNamespaceIndex,
		sNetID			:= '127.0.0.1.1.1',
		nPort			:= 851,
		nIndexGroup		:= 16#4020,
		nIndexOffset	:= 0,
		pOutputArgInfoAndData 	:= ADR(stADSReadRes),		// buffer for output argument info and output data
		cbOutputArgInfoAndData	:= SIZEOF(stADSReadRes),	// size output argument info + Data
		cbReadData		:= SIZEOF(stADSReadRes.nReadData),	//size of Data only
		nNumberOfOutputArguments:= nNumberOfOutputArguments,
		pOutputArgInfo	:= ADR(stOutputArgInfo),
		cbOutputArgInfo	:= SIZEOF(stOutputArgInfo)		
		);


	IF NOT fbUA_MethodCall_ADSReadReq.bBusy THEN
		fbUA_MethodCall_ADSReadReq(bExecute := FALSE);
		IF NOT fbUA_MethodCall_ADSReadReq.bError THEN
			(* session closed *)
			iState 		:= iState + 1; (* close session *)
		ELSE
			bError		:= TRUE;
			nErrorID	:= fbUA_MethodCall_ADSReadReq.nErrorID;
			iState 		:= 4; (* close session *)
		END_IF
	END_IF


4:	(* close session *)
	fbUA_Disconnect(
		Execute			:= TRUE,
		ConnectionHdl	:= nConnectionHdl
	);

	IF NOT fbUA_Disconnect.Busy THEN
		fbUA_Disconnect(Execute := FALSE);
		bBusy := FALSE;
		IF NOT fbUA_Disconnect.Error THEN
			(* session closed *)
			iState 		:= 0; (* idle *)
			IF NOT bError THEN 
				bDone 	:= TRUE;
			END_IF
		ELSE
			bError			:= TRUE;
			nErrorID		:= fbUA_Disconnect.ErrorID;
			iState 			:= 0; (* idle *)
			nConnectionHdl	:= 0;
		END_IF
	END_IF
END_CASE

END_PROGRAM

// ---- BECKHOFF SPECIFIC helper library/POUs/MethodCall/UA_MethodCall_ADSReadReq.TcPOU
FUNCTION_BLOCK UA_MethodCall_ADSReadReq
VAR_INPUT
	bExecute			: BOOL;
	nConnectionHdl		: DWORD;
	nNamespaceIndex		: UINT; 			(* to be retrieved using UA_GetNamespaceIndex *)
	sNetID				: T_AmsNetId; 		(* AmsNetId OF the Target *)
	nPort				: INT; 				(* Port number	*)
	nIndexGroup			: DINT;				(* IndexGroup*)
	nIndexOffset		: DINT; 			(* IndexOffset*)
	pOutputArgInfoAndData	: PVOID;
	cbOutputArgInfoAndData	: UDINT;			(* Count of bytes to be read*)
	cbReadData			: UDINT;			(* Count of bytes to be read*)
	nNumberOfOutputArguments	: UDINT; 
	pOutputArgInfo		: POINTER TO ST_UAMethodArgInfo; 
	cbOutputArgInfo		: UDINT;
	Timeout				: TIME := DEFAULT_ADS_TIMEOUT;
END_VAR
VAR_OUTPUT
	cbReadData_R		: UDINT;			(* Count of bytes to be read*)
	bDone				: BOOL;
	bBusy				: BOOL;
	bError				: BOOL;
	nErrorID			: DWORD;
END_VAR
VAR
	iReadReqState			: INT;
	RTrig					: R_TRIG;

	fbUA_MethodGetHandle	: UA_MethodGetHandle;
	nMethodHdl				: DWORD;
	ObjectNodeID			: ST_UANodeID;
	MethodNodeID			: ST_UANodeID;

	fbUA_MethodCall			: UA_MethodCall;
	InputArguments			: ARRAY [1..nNumberOfInputArguments] OF ST_UAMethodArgInfo; (*ReadReq has 5 input parameters *)
	
	nArg					: INT;
	fbUA_MethodReleaseHandle: UA_MethodReleaseHandle;

	nInputData			: ARRAY [1..nInputArgSize] OF BYTE; (* NetID(24)+ Port(2)+ IG(4)+ IO(4)+ cbData(4)*)
	nOffset				: UDINT;
	bInputDataError		: BOOL;
END_VAR
VAR CONSTANT
	nInputArgSize			: UDINT := 38; (* NetID(24)+ Port(2)+ IG(4)+ IO(4)+ cbData(4)*)
	nNumberOfInputArguments : UDINT := 5;
END_VAR

(*
ADSReadReq(
******** Input Arguments ********
	string24 sNetID, 		: AmsNetId of the Target
	int16 Port,			: Port number	
	int32 IndexGroup,		: IndexGroup
	int32 IndexOffset,		: IndexOffset
	uint32 cbData			: Count of bytes to be read
******** Output Arguments ********
	bytestring Data		: Data read from device
);

*)
RTrig(CLK:= bExecute);

CASE iReadReqState OF

0:	(* Get Method Handle *)
	IF RTrig.Q THEN
		bBusy	:= TRUE;
		bDone 	:= FALSE;
		bError	:= FALSE;
		nErrorID	:= 0;
		ObjectNodeID.eIdentifierType 	:= eUAIdentifierType_String;
		ObjectNodeID.nNamespaceIndex 	:= nNamespaceIndex;
		ObjectNodeID.sIdentifier		:= 'ADSAMS';
	
		MethodNodeID.eIdentifierType 	:= eUAIdentifierType_String;
		MethodNodeID.nNamespaceIndex 	:= nNamespaceIndex;
		MethodNodeID.sIdentifier		:= 'ADSAMS.AdsReadReq';

		M_Init();
		IF bInputDataError = FALSE THEN
			iReadReqState 	:= iReadReqState + 1;
		ELSE
			bBusy 		:= FALSE; 
			bError 		:= TRUE;
			nErrorID 	:= DEVICE_INVALIDSIZE; //16#705 parameter size not correct
		END_IF
		
	END_IF


1:	(* Method Get Handle *)
	fbUA_MethodGetHandle(
			Execute			:= TRUE,
			ConnectionHdl	:= nConnectionHdl,
			ObjectNodeID	:= ObjectNodeID,
			MethodNodeID 	:= MethodNodeID,
			Timeout			:= Timeout,
			MethodHdl		=> nMethodHdl
		);
	IF NOT fbUA_MethodGetHandle.Busy THEN
		fbUA_MethodGetHandle(Execute := FALSE);

		IF NOT fbUA_MethodGetHandle.Error THEN
			(*  *)
			iReadReqState 	:= iReadReqState + 1; (* Call Method *)
		ELSE
			bError		:= TRUE;
			nErrorID		:= fbUA_MethodGetHandle.ErrorID;
			iReadReqState 	:= 3; (* Release Handle *)
		END_IF
	END_IF


2:	(* Method Call *)
	fbUA_MethodCall(
		Execute					:= TRUE,
		ConnectionHdl			:= nConnectionHdl,
		MethodHdl				:= nMethodHdl,
		nNumberOfInputArguments := nNumberOfInputArguments, (* 5 *)
		pInputArgInfo			:= ADR(InputArguments),
		cbInputArgInfo			:= SIZEOF(InputArguments),
		pInputArgData			:= ADR(nInputData),
		cbInputArgData			:= nOffset,
		pInputWriteData			:= 0,		
		cbInputWriteData		:= 0,
		nNumberOfOutputArguments:= nNumberOfOutputArguments, (* input parameter: to be assigned by customer *)
		pOutputArgInfo			:= pOutputArgInfo,
		cbOutputArgInfo			:= cbOutputArgInfo,
		pOutputArgInfoAndData	:= pOutputArgInfoAndData,
		cbOutputArgInfoAndData	:= cbOutputArgInfoAndData,
		Timeout					:= Timeout
	);

	IF NOT fbUA_MethodCall.Busy THEN
		fbUA_MethodCall(Execute := FALSE, cbRead_R => cbReadData_R);

		IF NOT fbUA_MethodCall.Error THEN
			(*  *)
			iReadReqState 	:= iReadReqState + 1; (* Release handle *)
		ELSE
			bError		:= TRUE;
			nErrorID		:= fbUA_MethodCall.ErrorID;
			iReadReqState 	:= 3; (* Release handle *)
		END_IF
	END_IF


3:	(* Release Method Handle *)
	fbUA_MethodReleaseHandle(
		Execute			:= TRUE,
		ConnectionHdl	:= nConnectionHdl,
		MethodHdl		:= nMethodHdl,
		Timeout			:= Timeout
	);

	IF NOT fbUA_MethodReleaseHandle.Busy THEN
		fbUA_MethodReleaseHandle(Execute := FALSE);
		bBusy := FALSE;
		IF NOT fbUA_MethodReleaseHandle.Error THEN
			(* session closed *)
			bDone := TRUE;
			iReadReqState 	:= 0; (* idle *)
		ELSE
			bError			:= TRUE;
			nErrorID		:= fbUA_MethodReleaseHandle.ErrorID;
			iReadReqState 	:= 0; (* idle *)
		END_IF
	END_IF
END_CASE

ACTION M_Init:
bInputDataError := FALSE; 
nOffset := 0;
MEMSET(ADR(InputArguments),0,SIZEOF(InputArguments));
MEMSET(ADR(nInputData),0,SIZEOF(nInputData));

nArg := 1;
(*sNetID := sAmsNetID;*)		(********** NET ID **********)
InputArguments[nArg].DataType			:= eUAType_String;
InputArguments[nArg].ValueRank			:= -1; 							(* Scalar or Array *)
InputArguments[nArg].ArrayDimensions[1]	:= 0; 							(* Number of Dimension in case its an array *)
InputArguments[nArg].nLenData			:= INT_TO_UDINT(LEN(sNetId)) + 1;				(* Length if its a STRING *)
IF nOffset + INT_TO_UDINT(LEN(sNetId))+1 > nInputArgSize THEN 
	bInputDataError := TRUE;
	RETURN;
ELSE
	MEMCPY(ADR(nInputData)+nOffset,ADR(sNetId),INT_TO_UDINT(LEN(sNetId))+1);				(* VALUE in BYTES FORM *)
	nOffset := nOffset + INT_TO_UDINT(LEN(sNetId))+1;
END_IF

nArg := nArg + 1;
(* nPort := 851;*)			(********** PORT **********)
InputArguments[nArg].DataType			:= eUAType_Int16;
InputArguments[nArg].ValueRank			:= -1; 							(* Scalar or Array *)
InputArguments[nArg].ArrayDimensions[1]	:= 0; 							(* Number of Dimension in case its an array *)
InputArguments[nArg].nLenData			:= SIZEOF(nPort);				(* Length if its a STRING *)
IF nOffset + SIZEOF(nPort) > nInputArgSize THEN 
	bInputDataError := TRUE;
	RETURN;
ELSE
	MEMCPY(ADR(nInputData)+nOffset,ADR(nPort),SIZEOF(nPort));			(* VALUE in BYTES FORM *)
	nOffset := nOffset + SIZEOF(nPort);
END_IF

nArg := nArg + 1;
(*nIndexGroup := 16#4020;*)	(********** INDEX GROUP **********)
InputArguments[nArg].DataType			:= eUAType_Int32;
InputArguments[nArg].ValueRank			:= -1; 							(* Scalar or Array *)
InputArguments[nArg].ArrayDimensions[1]	:= 0; 							(* Number of Dimension in case its an array *)
InputArguments[nArg].nLenData			:= SIZEOF(nIndexGroup);			(* Length if its a STRING *)
IF nOffset + SIZEOF(nIndexGroup) > nInputArgSize THEN 
	bInputDataError := TRUE;
	RETURN;
ELSE
	MEMCPY(ADR(nInputData)+nOffset,ADR(nIndexGroup),SIZEOF(nIndexGroup));		(* VALUE in BYTES FORM *)
	nOffset := nOffset + SIZEOF(nIndexGroup);
END_IF

nArg := nArg + 1;
(*nIndexOffset := 0; *)		(********** INDEX OFFSET **********)
InputArguments[nArg].DataType			:= eUAType_Int32;
InputArguments[nArg].ValueRank			:= -1; 							(* Scalar or Array *)
InputArguments[nArg].ArrayDimensions[1]	:= 0; 							(* Number of Dimension in case its an array *)
InputArguments[nArg].nLenData			:= SIZEOF(nIndexOffset);		(* Length if its a STRING *)
IF nOffset + SIZEOF(nIndexOffset) > nInputArgSize THEN 
	bInputDataError := TRUE;
	RETURN;
ELSE
	MEMCPY(ADR(nInputData)+nOffset,ADR(nIndexOffset),SIZEOF(nIndexOffset));	(* VALUE in BYTES FORM *)
	nOffset := nOffset + SIZEOF(nIndexOffset);
END_IF

nArg := nArg + 1;
(*nReadLength := 2; *)		(*********** ReadLength ***********)
InputArguments[nArg].DataType			:= eUAType_UInt32;
InputArguments[nArg].ValueRank			:= -1; 							(* Scalar or Array *)
InputArguments[nArg].ArrayDimensions[1]	:= 0; 							(* Number of Dimension in case its an array *)
InputArguments[nArg].nLenData			:= SIZEOF(cbReadData);	
IF nOffset + SIZEOF(cbReadData) > nInputArgSize THEN 
	bInputDataError := TRUE;
	RETURN;
ELSE			(* Length if its a STRING *)
	MEMCPY(ADR(nInputData)+nOffset,ADR(cbReadData),SIZEOF(cbReadData));				(* VALUE in BYTES FORM *)
	nOffset := nOffset + SIZEOF(cbReadData);
END_IF
END_ACTION

END_FUNCTION_BLOCK

// ---- POUs/PRG_ADSWriteReq.TcPOU
PROGRAM PRG_ADSWriteReq
VAR
	fbUA_Connect			: UA_Connect;
	SessionConnectInfo		: ST_UASessionConnectInfo;
	sOpcUA_URL				: STRING(MAX_STRING_LENGTH);
	nConnectionHdl			: DWORD;

	fbUA_GetNamespaceIndex 	: UA_GetNamespaceIndex;
	nNamespaceIndex			: UINT;

	fbUA_NodeReleaseHandle	: UA_NodeReleaseHandle;
	
	fbUA_MethodCall_ADSWriteReq	: UA_MethodCall_ADSWriteReq;
	nWriteData	: INT := 2242;
	
	fbUA_Disconnect		: UA_Disconnect;
		
	bTest		: BOOL:= TRUE;
	bDone		: BOOL;
	bBusy		: BOOL;
	bError		: BOOL;
	nErrorID	: DWORD;
	iState		: INT;	
END_VAR


CASE iState OF
0:	(* idle *)
	IF bTest THEN
		bTest		:= FALSE;
		bError		:= FALSE;
		nErrorID	:= 0;

		(* Parameterize *)
		sOpcUA_URL						:= 'opc.tcp://localhost:4840';	(* OpcUA Url of the device with ip address *)

		SessionConnectInfo.tConnectTimeout 		:= T#1S;
		SessionConnectInfo.tSessionTimeout 		:= T#1S;
		SessionConnectInfo.sApplicationName		:= '';
//		SessionConnectInfo.sApplicationUri 		:= '';
		SessionConnectInfo.eSecurityMode 		:= eUASecurityMsgMode_None;
		SessionConnectInfo.eSecurityPolicyUri 	:= eUASecurityPolicy_None;
		SessionConnectInfo.eTransportProfileUri := eUATransportProfileUri_UATcp;

		iState	:= iState + 1;	(* open ua session *)
	END_IF

1:	(* open UA session *)
	fbUA_Connect(
		Execute				:= TRUE,
		ServerURL			:= sOpcUA_URL,
		SessionConnectInfo	:= SessionConnectInfo,
		Timeout				:= T#5S,
		ConnectionHdl		=> nConnectionHdl
	);

	IF NOT fbUA_Connect.Busy THEN
		fbUA_Connect(Execute := FALSE);

		IF NOT fbUA_Connect.Error THEN
			(* session open *)
			iState := iState + 1;	(* get namespace index *)
		ELSE
			bError			:= TRUE;
			nErrorID		:= fbUA_Connect.ErrorID;
			nConnectionHdl	:= 0;
			iState 			:= 0; (* idle *)
		END_IF
	END_IF


2:	(* GetNS Index *)
	fbUA_GetNamespaceIndex(
		Execute			:= TRUE,
		ConnectionHdl	:= nConnectionHdl,
		NamespaceUri	:= 'ADSAMS',
		NamespaceIndex	=> nNamespaceIndex
	);

	IF NOT fbUA_GetNamespaceIndex.Busy THEN
		fbUA_GetNamespaceIndex(Execute := FALSE);

		IF NOT fbUA_GetNamespaceIndex.Error THEN
			(* session closed *)
			iState 		:= iState + 1; (* method *)
		ELSE
			bError		:= TRUE;
			nErrorID	:= fbUA_GetNamespaceIndex.ErrorID;
			iState 		:= 4; (* close session *)
		END_IF
	END_IF

3:	(*  Method  *)
	fbUA_MethodCall_ADSWriteReq(
		bExecute		:= TRUE,
		nConnectionHdl	:= nConnectionHdl,
		nNamespaceIndex := nNamespaceIndex,
		sNetID			:= '127.0.0.1.1.1',
		nPort			:= 851,
		nIndexGroup		:= 16#4020,
		nIndexOffset	:= 0,
		pWriteData 		:= ADR(nWriteData),
		cbWriteData		:= SIZEOF(nWriteData)
		);


	IF NOT fbUA_MethodCall_ADSWriteReq.bBusy THEN
		fbUA_MethodCall_ADSWriteReq(bExecute := FALSE);
		IF NOT fbUA_MethodCall_ADSWriteReq.bError THEN
			(* session closed *)
			iState 		:= iState + 1; (* close session *)
		ELSE
			bError		:= TRUE;
			nErrorID	:= fbUA_MethodCall_ADSWriteReq.nErrorID;
			iState 		:= 4; (* close session *)
		END_IF
	END_IF


4:	(* close session *)
	fbUA_Disconnect(
		Execute			:= TRUE,
		ConnectionHdl	:= nConnectionHdl
	);

	IF NOT fbUA_Disconnect.Busy THEN
		fbUA_Disconnect(Execute := FALSE);
		bBusy := FALSE;
		IF NOT fbUA_Disconnect.Error THEN
			(* session closed *)
			iState 		:= 0; (* idle *)
			IF NOT bError THEN 
				bDone 	:= TRUE;
			END_IF
		ELSE
			bError			:= TRUE;
			nErrorID		:= fbUA_Disconnect.ErrorID;
			iState 			:= 0; (* idle *)
			nConnectionHdl	:= 0;
		END_IF
	END_IF
END_CASE

END_PROGRAM

// ---- BECKHOFF SPECIFIC helper library/POUs/MethodCall/UA_MethodCall_ADSWriteReq.TcPOU
FUNCTION_BLOCK UA_MethodCall_ADSWriteReq
VAR_INPUT
	bExecute			: BOOL;
	nConnectionHdl		: DWORD;
	nNamespaceIndex		: UINT; 			(* to be retrieved using UA_GetNamespaceIndex *)
	sNetID				: T_AmsNetId; 		(* AmsNetId OF the Target *)
	nPort				: INT; 			(* Port number	*)
	nIndexGroup			: DINT;			(* IndexGroup*)
	nIndexOffset		: DINT; 			(* IndexOffset*)
	pWriteData			: PVOID;
	cbWriteData			: UDINT;			(* Count of bytes to be written*)
	Timeout				: TIME := DEFAULT_ADS_TIMEOUT;
END_VAR
VAR_OUTPUT
	bDone				: BOOL;
	bBusy				: BOOL;
	bError				: BOOL;
	nErrorID			: DWORD;
END_VAR
VAR
	iWriteReqState		: INT;
	RTrig				: R_TRIG;

	fbUA_MethodGetHandle	: UA_MethodGetHandle;
	nMethodHdl				: DWORD;
	ObjectNodeID			: ST_UANodeID;
	MethodNodeID			: ST_UANodeID;

	fbUA_MethodCall			: UA_MethodCall;
	InputArguments			: ARRAY [1..nNumberOfInputArguments] OF ST_UAMethodArgInfo; (*WriteReq has 5 input parameters *)
	nNumberOfOutputArguments_R: UDINT;
	nArg					: INT;
	nInputData				: ARRAY [1..nInputArgSize] OF BYTE; (* NetID(24)+ Port(2)+ IG(4)+ IO(4)*)
	nOffset					: UDINT;


	fbUA_MethodReleaseHandle	: UA_MethodReleaseHandle; 
	bInputDataError				: BOOL;
END_VAR
VAR CONSTANT
	nInputArgSize				: UDINT := 34; // (* NetID(24)+ Port(2)+ IG(4)+ IO(4)*)
	nNumberOfInputArguments 	: UDINT := 5;
	nNumberOfOutputArguments	: UDINT := 0;
END_VAR

(*
ADSWriteReq(
******** Input Arguments ********
	string sNetID, 		: AmsNetId of the Target
	int16 Port,			: Port number	
	int32 IndexGroup,	: IndexGroup
	int32 IndexOffset,	: IndexOffset
	byteString Data		: Data to be written to the device
******** Output Arguments ********
);
*)

RTrig(CLK:= bExecute);

CASE iWriteReqState OF

0:	(* Get Method Handle *)
	IF RTrig.Q THEN
		bBusy		:= TRUE;
		bDone 		:= FALSE;
		bError		:= FALSE;
		nErrorID	:= 0;
		ObjectNodeID.eIdentifierType 	:= eUAIdentifierType_String;
		ObjectNodeID.nNamespaceIndex 	:= nNamespaceIndex;
		ObjectNodeID.sIdentifier		:= 'ADSAMS';
	
		MethodNodeID.eIdentifierType 	:= eUAIdentifierType_String;
		MethodNodeID.nNamespaceIndex 	:= nNamespaceIndex;
		MethodNodeID.sIdentifier		:= 'ADSAMS.AdsWriteReq';

		M_Init();
		IF bInputDataError = FALSE THEN
			iWriteReqState 	:= iWriteReqState + 1;
		ELSE
			bBusy		:= FALSE;
			bError 		:= TRUE;
			nErrorID 	:= DEVICE_INVALIDSIZE; //16#705 parameter size not correct
		END_IF
	END_IF


1:	(* Method Get Handle *)
	fbUA_MethodGetHandle(
			Execute			:= TRUE,
			ConnectionHdl	:= nConnectionHdl,
			ObjectNodeID	:= ObjectNodeID,
			MethodNodeID 	:= MethodNodeID,
			Timeout			:= Timeout,
			MethodHdl		=> nMethodHdl
		);
	IF NOT fbUA_MethodGetHandle.Busy THEN
		fbUA_MethodGetHandle(Execute := FALSE);

		IF NOT fbUA_MethodGetHandle.Error THEN
			(*  *)
			iWriteReqState 	:= iWriteReqState + 1; (* Call Method *)
		ELSE
			bError			:= TRUE;
			nErrorID		:= fbUA_MethodGetHandle.ErrorID;
			iWriteReqState 	:= 3; (* Release Handle *)
		END_IF
	END_IF


2:	(* Method Call *)
	fbUA_MethodCall(
		Execute					:= TRUE,
		ConnectionHdl			:= nConnectionHdl,
		MethodHdl				:= nMethodHdl,
		nNumberOfInputArguments := nNumberOfInputArguments,		(* 5 *)
		pInputArgInfo			:= ADR(InputArguments),
		cbInputArgInfo			:= SIZEOF(InputArguments),
		pInputArgData			:= ADR(nInputData),
		cbInputArgData			:= nOffset,
		pInputWriteData			:= pWriteData,
		cbInputWriteData		:= cbWriteData,
		nNumberOfOutputArguments:= nNumberOfOutputArguments,		(* 0 *)
		pOutputArgInfo			:= 0,
		cbOutputArgInfo			:= 0,
		pOutputArgInfoAndData	:= ADR(nNumberOfOutputArguments_R),
		cbOutputArgInfoAndData	:= SIZEOF(nNumberOfOutputArguments_R),
		Timeout					:= Timeout
	);

	IF NOT fbUA_MethodCall.Busy THEN
		fbUA_MethodCall(Execute := FALSE);
		IF NOT fbUA_MethodCall.Error THEN
			(*  *)
			iWriteReqState 	:= iWriteReqState + 1; (* Release handle *)
			(*MEMSET(ADR(Data),0,nMaxNumberofOutputArgBytes);
			MEMCPY(ADR(Data),ADR(OutputArguments),cbData); *)
		ELSE
			bError			:= TRUE;
			nErrorID		:= fbUA_MethodCall.ErrorID;
			iWriteReqState	:= 3; (* Release handle *)
		END_IF
	END_IF


3:	(* Release Method Handle *)
	fbUA_MethodReleaseHandle(
		Execute			:= TRUE,
		ConnectionHdl	:= nConnectionHdl,
		MethodHdl		:= nMethodHdl,
		Timeout			:= Timeout
	);

	IF NOT fbUA_MethodReleaseHandle.Busy THEN
		fbUA_MethodReleaseHandle(Execute := FALSE);
		bBusy := FALSE;
		IF NOT fbUA_MethodReleaseHandle.Error THEN
			(* session closed *)
			bDone := TRUE;
			iWriteReqState 	:= 0; (* idle *)
		ELSE
			bError			:= TRUE;
			nErrorID		:= fbUA_MethodReleaseHandle.ErrorID;
			iWriteReqState 	:= 0; (* idle *)
		END_IF
	END_IF
END_CASE

ACTION M_Init:
bInputDataError := FALSE; 
nOffset := 0;
MEMSET(ADR(InputArguments),0,SIZEOF(InputArguments));
MEMSET(ADR(nInputData),0,SIZEOF(nInputData));

nArg := 1;
(*sNetID := sAmsNetID;*)	(********** NET ID **********);
InputArguments[nArg].DataType			:= eUAType_String;
InputArguments[nArg].ValueRank			:= -1; 							(* Scalar = -1 or Array *)
InputArguments[nArg].ArrayDimensions[1]	:= 0; 							(* Number of Dimension in case its an array *)
InputArguments[nArg].nLenData			:= INT_TO_UDINT(LEN(sNetId)) + 1;				(* Length if its a STRING *)
IF nOffset + INT_TO_UDINT(LEN(sNetId))+1 > nInputArgSize THEN 
	bInputDataError := TRUE;
	RETURN;
ELSE
	MEMCPY(ADR(nInputData)+nOffset,ADR(sNetId),INT_TO_UDINT(LEN(sNetId))+1);				(* VALUE in BYTES FORM *)
	nOffset := nOffset + INT_TO_UDINT(LEN(sNetId))+1;
END_IF

nArg := nArg + 1;
(* nPort := 851;*)			(********** PORT **********)
InputArguments[nArg].DataType			:= eUAType_Int16;
InputArguments[nArg].ValueRank			:= -1; 							(* Scalar = -1 or Array *)
InputArguments[nArg].ArrayDimensions[1]	:= 0; 							(* Number of Dimension in case its an array *)
InputArguments[nArg].nLenData			:= SIZEOF(nPort);				(* Length if its a STRING *)
IF nOffset + SIZEOF(nPort) > nInputArgSize THEN 
	bInputDataError := TRUE;
	RETURN;
ELSE
	MEMCPY(ADR(nInputData)+nOffset,ADR(nPort),SIZEOF(nPort));			(* VALUE in BYTES FORM *)
	nOffset := nOffset + SIZEOF(nPort);
END_IF

nArg := nArg + 1;
(*nIndexGroup := 16#4020;*)	(********** INDEX GROUP **********)
InputArguments[nArg].DataType			:= eUAType_Int32;
InputArguments[nArg].ValueRank			:= -1; 							(* Scalar = -1 or Array *)
InputArguments[nArg].ArrayDimensions[1]	:= 0; 							(* Number of Dimension in case its an array *)
InputArguments[nArg].nLenData			:= SIZEOF(nIndexGroup);			(* Length if its a STRING *)
IF nOffset + SIZEOF(nIndexGroup) > nInputArgSize THEN 
	bInputDataError := TRUE;
	RETURN;
ELSE
	MEMCPY(ADR(nInputData)+nOffset,ADR(nIndexGroup),SIZEOF(nIndexGroup));		(* VALUE in BYTES FORM *)
	nOffset := nOffset + SIZEOF(nIndexGroup);
END_IF

nArg := nArg + 1;
(*nIndexOffset := 0; *)		(********** INDEX OFFSET **********)
InputArguments[nArg].DataType			:= eUAType_Int32;
InputArguments[nArg].ValueRank			:= -1; 							(* Scalar = -1 or Array *)
InputArguments[nArg].ArrayDimensions[1]	:= 0; 							(* Number of Dimension in case its an array *)
InputArguments[nArg].nLenData			:= SIZEOF(nIndexOffset);		(* Length if its a STRING *)
IF nOffset + SIZEOF(nIndexOffset) > nInputArgSize THEN 
	bInputDataError := TRUE;
	RETURN;
ELSE
	MEMCPY(ADR(nInputData)+nOffset,ADR(nIndexOffset),SIZEOF(nIndexOffset));	(* VALUE in BYTES FORM *)
	nOffset := nOffset + SIZEOF(nIndexOffset);
END_IF

nArg := nArg + 1;
(*Data := 2; *)		(*********** WriteData ***********)
InputArguments[nArg].DataType			:= eUAType_ByteString;
InputArguments[nArg].ValueRank			:= -1; 							(* Scalar = -1 or Array *)
InputArguments[nArg].ArrayDimensions[1]	:= 0; 							(* Number of Dimension in case its an array *)
InputArguments[nArg].nLenData			:= cbWriteData;
END_ACTION

END_FUNCTION_BLOCK

// ---- POUs/PRG_ADSReadDeviceInfoReq.TcPOU
PROGRAM PRG_ADSReadDeviceInfoReq
VAR
	fbUA_Connect			: UA_Connect;
	SessionConnectInfo		: ST_UASessionConnectInfo;
	sOpcUA_URL				: STRING(MAX_STRING_LENGTH);
	nConnectionHdl			: DWORD;

	fbUA_GetNamespaceIndex 	: UA_GetNamespaceIndex;
	nNamespaceIndex			: UINT;

	fbUA_NodeReleaseHandle	: UA_NodeReleaseHandle;
	
	fbUA_MethodCall_ADSReadDeviceInfo	: UA_MethodCall_ADSReadDeviceInfoReq;
	sDeviceName			: STRING(19);	(* DeviceName *)
	nVersion			: SINT;			(* Version *)
	nRevision			: SINT;			(* Revision *)
	nBuild				: INT;			(* Build *)
	
	fbUA_Disconnect		: UA_Disconnect;
		
	bTest		: BOOL := TRUE;
	bDone		: BOOL;
	bBusy		: BOOL;
	bError		: BOOL;
	nErrorID	: DWORD;
	iState		: INT;	
END_VAR


CASE iState OF
0:	(* idle *)
	IF bTest THEN
		bTest	:= FALSE;
		bError	:= FALSE;
		nErrorID	:= 0;

		(* Parameterize *)
		sOpcUA_URL						:= 'opc.tcp://localhost:4840';	(* OpcUA Url of the device with ip address *)

		SessionConnectInfo.tConnectTimeout 		:= T#1S;
		SessionConnectInfo.tSessionTimeout 		:= T#1S;
		SessionConnectInfo.sApplicationName		:= '';
//		SessionConnectInfo.sApplicationUri 		:= '';
		SessionConnectInfo.eSecurityMode 		:= eUASecurityMsgMode_None;
		SessionConnectInfo.eSecurityPolicyUri 	:= eUASecurityPolicy_None;
		SessionConnectInfo.eTransportProfileUri := eUATransportProfileUri_UATcp;

		iState	:= iState + 1;	(* open ua session *)
	END_IF

1:	(* open UA session *)
	fbUA_Connect(
		Execute				:= TRUE,
		ServerURL			:= sOpcUA_URL,
		SessionConnectInfo	:= SessionConnectInfo,
		Timeout				:= T#5S,
		ConnectionHdl		=> nConnectionHdl
	);

	IF NOT fbUA_Connect.Busy THEN
		fbUA_Connect(Execute := FALSE);

		IF NOT fbUA_Connect.Error THEN
			(* session open *)
			iState := iState + 1;	(* get namespace index *)
		ELSE
			bError			:= TRUE;
			nErrorID		:= fbUA_Connect.ErrorID;
			nConnectionHdl	:= 0;
			iState 			:= 0; (* idle *)
		END_IF
	END_IF


2:	(* GetNS Index *)
	fbUA_GetNamespaceIndex(
		Execute			:= TRUE,
		ConnectionHdl	:= nConnectionHdl,
		NamespaceUri	:= 'ADSAMS',
		NamespaceIndex	=> nNamespaceIndex
	);

	IF NOT fbUA_GetNamespaceIndex.Busy THEN
		fbUA_GetNamespaceIndex(Execute := FALSE);

		IF NOT fbUA_GetNamespaceIndex.Error THEN
			(* session closed *)
			iState 		:= iState + 1; (* method *)
		ELSE
			bError		:= TRUE;
			nErrorID	:= fbUA_GetNamespaceIndex.ErrorID;
			iState 		:= 4; (* close session *)
		END_IF
	END_IF

3:	(*  Method  *)
	fbUA_MethodCall_ADSReadDeviceInfo(
		bExecute		:= TRUE,
		nConnectionHdl	:= nConnectionHdl,
		nNamespaceIndex	:= nNamespaceIndex,
		sNetID			:= '127.0.0.1.1.1',
		nPort			:= 10000,
		sDeviceName		=> sDeviceName,		(* ADS state *)
		nVersion		=> nVersion,			(* Device state *)
		nRevision		=> nRevision,
		nBuild			=> nBuild
		);


	IF NOT fbUA_MethodCall_ADSReadDeviceInfo.bBusy THEN
		fbUA_MethodCall_ADSReadDeviceInfo(	bExecute 	:= FALSE, 
											sDeviceName	=> sDeviceName,		(* ADS state *)
											nVersion	=> nVersion,			(* Device state *)
											nRevision	=> nRevision,
											nBuild		=> nBuild);
		IF NOT fbUA_MethodCall_ADSReadDeviceInfo.bError THEN
			(* session closed *)
			iState 		:= iState + 1; (* close session *)
		ELSE
			bError		:= TRUE;
			nErrorID	:= fbUA_MethodCall_ADSReadDeviceInfo.nErrorID;
			iState 		:= 4; (* close session *)
		END_IF
	END_IF


4:	(* close session *)
	fbUA_Disconnect(
		Execute			:= TRUE,
		ConnectionHdl	:= nConnectionHdl
	);

	IF NOT fbUA_Disconnect.Busy THEN
		fbUA_Disconnect(Execute := FALSE);
		bBusy := FALSE;
		IF NOT fbUA_Disconnect.Error THEN
			(* session closed *)
			iState 		:= 0; (* idle *)
			IF NOT bError THEN 
				bDone 	:= TRUE;
			END_IF
		ELSE
			bError			:= TRUE;
			nErrorID		:= fbUA_Disconnect.ErrorID;
			iState 			:= 0; (* idle *)
			nConnectionHdl	:= 0;
		END_IF
	END_IF
END_CASE

END_PROGRAM

// ---- BECKHOFF SPECIFIC helper library/POUs/MethodCall/UA_MethodCall_ADSReadDeviceInfoReq.TcPOU
FUNCTION_BLOCK UA_MethodCall_ADSReadDeviceInfoReq
VAR_INPUT
	bExecute			: BOOL;
	nConnectionHdl		: DWORD;
	nNamespaceIndex		: UINT; 			(* to be retrieved using UA_GetNamespaceIndex *)
	sNetID				: T_AmsNetId; 		(* AmsNetId OF the Target *)
	nPort				: INT; 				(* Port number	*)
	Timeout				: TIME := DEFAULT_ADS_TIMEOUT;
END_VAR
VAR_OUTPUT
	sDeviceName			: STRING(19);	(* DeviceName *)
	nVersion			: SINT;			(* Version *)
	nRevision			: SINT;			(* Revision *)
	nBuild				: INT;			(* Build *)
	cbReadData_R		: UDINT; 
	bDone				: BOOL;
	bBusy				: BOOL;
	bError				: BOOL;
	nErrorID			: DWORD;
END_VAR
VAR
	iReadDeviceInfoState	: INT;
	RTrig					: R_TRIG;

	fbUA_MethodGetHandle	: UA_MethodGetHandle;
	nMethodHdl				: DWORD;
	ObjectNodeID			: ST_UANodeID;
	MethodNodeID			: ST_UANodeID;

	fbUA_MethodCall			: UA_MethodCall;
	InputArguments			: ARRAY [1..nNumberOfInputArguments] OF ST_UAMethodArgInfo; (*ReadDeviceInfoReq has 2 input parameters *)
	stOutputArgInfoAndData	: ST_UAMethodCall_AdsReadDeviceInfoRes;
	
	nArg					: INT;
	stOutputArgInfo			: ARRAY [1..nNumberOfOutputArguments] OF ST_UAMethodArgInfo;
	
	fbUA_MethodReleaseHandle	: UA_MethodReleaseHandle;

	nInputData			: ARRAY [1..nInputArgSize] OF BYTE; (* NetID (24) + Port (2) *)
	nOffset				: UDINT;
	nOffsetOutputData	: UDINT := 0; 
	bInputDataError		: BOOL; 
END_VAR
VAR CONSTANT
	nInputArgSize				: UDINT := 26; (* NetID (24) + Port (2) *)
	nNumberOfInputArguments 	: UDINT := 2;
	nNumberOfOutputArguments 	: UDINT := 4;
END_VAR

(*
ADSReadDeviceInfoReq(
******** Input Arguments ********
	string sNetID, 		: AmsNetId of the Target
	int16 Port,			: Port number	
	
******** Output Arguments ********
	string DeviceName,		: Device name
	byte Version,			: Version
	byte Revision			: Revision
	int16 Build			: Build
);
*)
RTrig(CLK:= bExecute);

CASE iReadDeviceInfoState OF

0:	(* Get Method Handle *)
	IF RTrig.Q THEN
		bInputDataError := FALSE; 
		bBusy		:= TRUE;
		bDone 		:= FALSE;
		bError		:= FALSE;
		nErrorID	:= 0;
		ObjectNodeID.eIdentifierType 	:= eUAIdentifierType_String;
		ObjectNodeID.nNamespaceIndex 	:= nNamespaceIndex;
		ObjectNodeID.sIdentifier		:= 'ADSAMS';
	
		MethodNodeID.eIdentifierType 	:= eUAIdentifierType_String;
		MethodNodeID.nNamespaceIndex 	:= nNamespaceIndex;
		MethodNodeID.sIdentifier		:= 'ADSAMS.AdsReadDeviceInfoReq';

		M_Init();
		IF bInputDataError = FALSE THEN
			iReadDeviceInfoState 	:= iReadDeviceInfoState + 1;
		ELSE
			bBusy 		:= FALSE; 
			bError 		:= TRUE;
			nErrorID 	:= DEVICE_INVALIDSIZE; //16#705 parameter size not correct
		END_IF
		sDeviceName		:= '';		(* ADS state *)
		nVersion		:= 0;		(* Device state *)
		nRevision		:= 0;
		nBuild			:= 0;
	END_IF


1:	(* Method Get Handle *)
	fbUA_MethodGetHandle(
			Execute			:= TRUE,
			ConnectionHdl	:= nConnectionHdl,
			ObjectNodeID	:= ObjectNodeID,
			MethodNodeID 	:= MethodNodeID,
			Timeout			:= Timeout,
			MethodHdl		=> nMethodHdl
		);
	IF NOT fbUA_MethodGetHandle.Busy THEN
		fbUA_MethodGetHandle(Execute := FALSE);

		IF NOT fbUA_MethodGetHandle.Error THEN
			(*  *)
			iReadDeviceInfoState 	:= iReadDeviceInfoState + 1; (* Call Method *)
		ELSE
			bError				:= TRUE;
			nErrorID			:= fbUA_MethodGetHandle.ErrorID;
			iReadDeviceInfoState:= 3; (* Release Handle *)
		END_IF
	END_IF


2:	(* Method Call *)
	fbUA_MethodCall(
		Execute					:= TRUE,
		ConnectionHdl			:= nConnectionHdl,
		MethodHdl				:= nMethodHdl,
		nNumberOfInputArguments := nNumberOfInputArguments,		(* 6 *)
		pInputArgInfo			:= ADR(InputArguments),
		cbInputArgInfo			:= SIZEOF(InputArguments),
		pInputArgData			:= ADR(nInputData),
		cbInputArgData			:= nOffset,
		pInputWriteData			:= 0,
		cbInputWriteData		:= 0,
		nNumberOfOutputArguments:= nNumberOfOutputArguments,	(* 4 *)
		pOutputArgInfo			:= ADR(stOutputArgInfo),
		cbOutputArgInfo			:= SIZEOF(stOutputArgInfo),
		pOutputArgInfoAndData	:= ADR(stOutputArgInfoAndData),
		cbOutputArgInfoAndData	:= SIZEOF(stOutputArgInfoAndData),
		Timeout					:= Timeout
	);
	IF NOT fbUA_MethodCall.Busy THEN
		fbUA_MethodCall(Execute := FALSE, cbRead_R => cbReadData_R);
		nOffsetOutputData := 0; 
		IF NOT fbUA_MethodCall.Error THEN
			(*  *)
			iReadDeviceInfoState:= iReadDeviceInfoState + 1; (* Release handle *)
			sDeviceName 		:= stOutputArgInfoAndData.stDeviceInfo.sDeviceName;
			nVersion   			:= stOutputArgInfoAndData.stDeviceInfo.nVersion;
			nRevision  			:= stOutputArgInfoAndData.stDeviceInfo.nRevision;
			nBuild     			:= stOutputArgInfoAndData.stDeviceInfo.nBuild;
		ELSE
			bError		:= TRUE;
			nErrorID	:= fbUA_MethodCall.ErrorID;
			iReadDeviceInfoState:= 3; (* Release handle *)
		END_IF
	END_IF


3:	(* Release Method Handle *)
	fbUA_MethodReleaseHandle(
		Execute			:= TRUE,
		ConnectionHdl	:= nConnectionHdl,
		MethodHdl		:= nMethodHdl,
		Timeout			:= Timeout
	);

	IF NOT fbUA_MethodReleaseHandle.Busy THEN
		fbUA_MethodReleaseHandle(Execute := FALSE);
		bBusy := FALSE;
		IF NOT fbUA_MethodReleaseHandle.Error THEN
			(* session closed *)
			bDone := TRUE;
			iReadDeviceInfoState 	:= 0; (* idle *)
		ELSE
			bError				:= TRUE;
			nErrorID			:= fbUA_MethodReleaseHandle.ErrorID;
			iReadDeviceInfoState:= 0; (* idle *)
		END_IF
	END_IF
END_CASE

ACTION M_Init:
bInputDataError := FALSE; 
nOffset := 0;
MEMSET(ADR(InputArguments),0,SIZEOF(InputArguments));
MEMSET(ADR(nInputData),0,SIZEOF(nInputData));

nArg := 1;
(*sNetID := sAmsNetID;*)	(********** NET ID **********)
InputArguments[nArg].DataType			:= eUAType_String;
InputArguments[nArg].ValueRank			:= -1; 						(* Scalar = -1 or Array *)
InputArguments[nArg].ArrayDimensions[1]	:= 0; 						(* Number of Dimension in case its an array *)
InputArguments[nArg].nLenData			:= INT_TO_UDINT(LEN(sNetId)) + 1;			(* Length if its a STRING *)
IF nOffset + INT_TO_UDINT(LEN(sNetId))+1 > nInputArgSize THEN 
	bInputDataError := TRUE;
	RETURN;
ELSE
	MEMCPY(ADR(nInputData)+nOffset,ADR(sNetId),INT_TO_UDINT(LEN(sNetId))+1);				(* VALUE in BYTES FORM *)
	nOffset := nOffset + INT_TO_UDINT(LEN(sNetId))+1;
END_IF

nArg := nArg + 1;
(* nPort := 851;*)			(********** PORT **********)
InputArguments[nArg].DataType			:= eUAType_Int16;
InputArguments[nArg].ValueRank			:= -1; 						(* Scalar = -1 or Array *)
InputArguments[nArg].ArrayDimensions[1]	:= 0; 						(* Number of Dimension in case its an array *)
InputArguments[nArg].nLenData			:= SIZEOF(nPort);			(* Length if its a STRING *)
IF nOffset + SIZEOF(nPort) > nInputArgSize THEN 
	bInputDataError := TRUE;
	RETURN;
ELSE
	MEMCPY(ADR(nInputData)+nOffset,ADR(nPort),SIZEOF(nPort));			(* VALUE in BYTES FORM *)
	nOffset := nOffset + SIZEOF(nPort);
END_IF

//************** Prepare Output Argument information ***********
stOutputArgInfo[1].nLenData := SIZEOF(sDeviceName);
stOutputArgInfo[2].nLenData := SIZEOF(nVersion); 
stOutputArgInfo[3].nLenData := SIZEOF(nRevision);
stOutputArgInfo[4].nLenData := SIZEOF(nBuild);
END_ACTION

END_FUNCTION_BLOCK

// ---- POUs/PRG_ADSReadStateReq.TcPOU
PROGRAM PRG_ADSReadStateReq
VAR
	fbUA_Connect			: UA_Connect;
	SessionConnectInfo		: ST_UASessionConnectInfo;
	sOpcUA_URL				: STRING(MAX_STRING_LENGTH);
	nConnectionHdl			: DWORD;

	fbUA_GetNamespaceIndex 	: UA_GetNamespaceIndex;
	nNamespaceIndex			: UINT;

	fbUA_NodeReleaseHandle	: UA_NodeReleaseHandle;
	
	fbUA_MethodCall_ADSReadStateReq		: UA_MethodCall_ADSReadStateReq;
	nAdsState			: DINT;			(* ADS state *)
	nDeviceState		: DINT;			(* Device state *)
	
	fbUA_Disconnect		: UA_Disconnect;
		
	bTest		: BOOL:= TRUE;
	bDone		: BOOL;
	bBusy		: BOOL;
	bError		: BOOL;
	nErrorID	: DWORD;
	iState		: INT;
END_VAR


CASE iState OF
0:	(* idle *)
	IF bTest THEN
		bTest	:= FALSE;
		bError	:= FALSE;
		nErrorID	:= 0;

		(* Parameterize *)
		sOpcUA_URL						:= 'opc.tcp://Pujak-nb:4840';	(* OpcUA Url of the device with ip address *)

		SessionConnectInfo.tConnectTimeout 	:= t#1s;
		SessionConnectInfo.tSessionTimeout 	:= t#1s;
		SessionConnectInfo.sApplicationName	:= '';
//		SessionConnectInfo.sApplicationUri 	:= '';
		SessionConnectInfo.eSecurityMode 		:= eUASecurityMsgMode_None;
		SessionConnectInfo.eSecurityPolicyUri 	:= eUASecurityPolicy_None;
		SessionConnectInfo.eTransportProfileUri := eUATransportProfileUri_UATcp;

		iState	:= iState + 1;	(* open ua session *)
	END_IF

1:	(* open UA session *)
	fbUA_Connect(
		Execute				:= TRUE,
		ServerURL			:= sOpcUA_URL,
		SessionConnectInfo	:= SessionConnectInfo,
		Timeout				:= T#5S,
		ConnectionHdl		=> nConnectionHdl
	);

	IF NOT fbUA_Connect.Busy THEN
		fbUA_Connect(Execute := FALSE);

		IF NOT fbUA_Connect.Error THEN
			(* session open *)
			iState := iState + 1;	(* get namespace index *)
		ELSE
			bError			:= TRUE;
			nErrorID		:= fbUA_Connect.ErrorID;
			nConnectionHdl	:= 0;
			iState 			:= 0; (* idle *)
		END_IF
	END_IF


2:	(* GetNS Index *)
	fbUA_GetNamespaceIndex(
		Execute			:= TRUE,
		ConnectionHdl	:= nConnectionHdl,
		NamespaceUri	:= 'ADSAMS',
		NamespaceIndex	=> nNamespaceIndex
	);

	IF NOT fbUA_GetNamespaceIndex.Busy THEN
		fbUA_GetNamespaceIndex(Execute := FALSE);

		IF NOT fbUA_GetNamespaceIndex.Error THEN
			(* session closed *)
			iState 		:= iState + 1; (* method *)
		ELSE
			bError		:= TRUE;
			nErrorID	:= fbUA_GetNamespaceIndex.ErrorID;
			iState 		:= 4; (* close session *)
		END_IF
	END_IF

3:	(*  Method  *)
	fbUA_MethodCall_ADSReadStateReq(
		bExecute		:= TRUE,
		nConnectionHdl	:= nConnectionHdl,
		nNamespaceIndex	:= nNamespaceIndex,
		sNetID			:= '127.0.0.1.1.1',
		nPort			:= 851 );
	IF NOT fbUA_MethodCall_ADSReadStateReq.bBusy THEN
		fbUA_MethodCall_ADSReadStateReq(	bExecute 	 := FALSE, 
											nAdsState	 => nAdsState,		(* Ads State *)
											nDeviceState => nDeviceState);
		IF NOT fbUA_MethodCall_ADSReadStateReq.bError THEN
			(* session closed *)
			iState 		:= iState + 1; (* close session *)
		ELSE
			bError		:= TRUE;
			nErrorID	:= fbUA_MethodCall_ADSReadStateReq.nErrorID;
			iState 		:= 4; (* close session *)
		END_IF
	END_IF


4:	(* close session *)
	fbUA_Disconnect(
		Execute			:= TRUE,
		ConnectionHdl	:= nConnectionHdl
	);

	IF NOT fbUA_Disconnect.Busy THEN
		fbUA_Disconnect(Execute := FALSE);
		bBusy := FALSE; 
		IF NOT fbUA_Disconnect.Error THEN
			(* session closed *)
			iState 		:= 0; (* idle *)
			IF NOT bError THEN 
				bDone 	:= TRUE;
			END_IF
		ELSE
			bError			:= TRUE;
			nErrorID		:= fbUA_Disconnect.ErrorID;
			iState 			:= 0; (* idle *)
			nConnectionHdl	:= 0;
		END_IF
	END_IF
END_CASE

END_PROGRAM

// ---- BECKHOFF SPECIFIC helper library/POUs/MethodCall/UA_MethodCall_ADSReadStateReq.TcPOU
FUNCTION_BLOCK UA_MethodCall_ADSReadStateReq
VAR_INPUT
	bExecute			: BOOL;
	nConnectionHdl		: DWORD;
	nNamespaceIndex		: UINT; 			(* to be retrieved using UA_GetNamespaceIndex *)
	sNetID				: T_AmsNetId; 		(* AmsNetId OF the Target *)
	nPort				: INT; 			(* Port number	*)
	cbData				: UDINT;			(* Count OF bytes to be read*)
	pData				: PVOID;
	Timeout				: TIME := DEFAULT_ADS_TIMEOUT;
END_VAR
VAR_OUTPUT
	nAdsState			: DINT;			(* ADS state *)
	nDeviceState		: DINT;			(* Device state *)
	cbReadData_R		: UDINT; 
	bDone				: BOOL;
	bBusy				: BOOL;
	bError				: BOOL;
	nErrorID			: DWORD;
END_VAR
VAR
	iReadStateReqState	: INT;
	RTrig				: R_TRIG;

	fbUA_MethodGetHandle: UA_MethodGetHandle;
	nMethodHdl			: DWORD;
	ObjectNodeID		: ST_UANodeID;
	MethodNodeID		: ST_UANodeID;

	fbUA_MethodCall		: UA_MethodCall;
	InputArguments		: ARRAY [1..nNumberOfInputArguments] OF ST_UAMethodArgInfo; (*ReadStateReq has 2 input parameters *)
	stOutputArgInfoAndData	: ST_UAMethodCall_AdsReadStateRes; // (4+OutputArgInfo+8)bytes
	stOutputArgInfo		: ARRAY [1..nNumberOfOutputArguments] OF ST_UAMethodArgInfo;
	
	nArg				: INT;
	nInputData			: ARRAY [1..nInputArgSize] OF BYTE; (* NetID(24) + Port(2) *)
	nOffset				: UDINT;
	
	fbUA_MethodReleaseHandle	: UA_MethodReleaseHandle;
	bInputDataError 			: BOOL;
END_VAR
VAR CONSTANT
	nInputArgSize				: UDINT := 26; (* NetID(24) + Port(2) *)
	nNumberOfInputArguments 	: UDINT := 2;
	nNumberOfOutputArguments	: UDINT := 3;
END_VAR

(*
ADSReadStateReq(
******** Input Arguments ********
	string sNetID, 		: AmsNetId of the Target
	int16 Port,			: Port number	
	
******** Output Arguments ********
	int32 AdsState,		: Ads State
	int32 DeviceState	: Device State
	ByteString Data		: Data
);
*)


RTrig(CLK:= bExecute);

CASE iReadStateReqState OF

0:	(* Get Method Handle *)
	IF RTrig.Q THEN
		bBusy	:= TRUE;
		bDone 	:= FALSE;
		bError	:= FALSE;
		nErrorID	:= 0;
		ObjectNodeID.eIdentifierType 	:= eUAIdentifierType_String;
		ObjectNodeID.nNamespaceIndex 	:= nNamespaceIndex;
		ObjectNodeID.sIdentifier		:= 'ADSAMS';
	
		MethodNodeID.eIdentifierType 	:= eUAIdentifierType_String;
		MethodNodeID.nNamespaceIndex 	:= nNamespaceIndex;
		MethodNodeID.sIdentifier		:= 'ADSAMS.AdsReadStateReq';
		
		M_Init();
		IF bInputDataError = FALSE THEN
			iReadStateReqState 	:= iReadStateReqState + 1;
		ELSE
			bBusy 		:= FALSE; 
			bError 		:= TRUE;
			nErrorID 	:= DEVICE_INVALIDSIZE; //16#705 parameter size not correct
		END_IF
		nAdsState		:= 0;			(* ADS state *)
		nDeviceState	:= 0;			(* Device state *)
	END_IF


1:	(* Method Get Handle *)
	fbUA_MethodGetHandle(
			Execute			:= TRUE,
			ConnectionHdl	:= nConnectionHdl,
			ObjectNodeID	:= ObjectNodeID,
			MethodNodeID 	:= MethodNodeID,
			Timeout			:= Timeout,
			MethodHdl		=> nMethodHdl
		);
	IF NOT fbUA_MethodGetHandle.Busy THEN
		fbUA_MethodGetHandle(Execute := FALSE);

		IF NOT fbUA_MethodGetHandle.Error THEN
			(*  *)
			iReadStateReqState 	:= iReadStateReqState + 1; (* Call Method *)
		ELSE
			bError				:= TRUE;
			nErrorID			:= fbUA_MethodGetHandle.ErrorID;
			iReadStateReqState 	:= 3; (* Release Handle *)
		END_IF
	END_IF


2:	(* Method Call *)
	fbUA_MethodCall(
		Execute					:= TRUE,
		ConnectionHdl			:= nConnectionHdl,
		MethodHdl				:= nMethodHdl,
		nNumberOfInputArguments := nNumberOfInputArguments,		(* 2 *)
		pInputArgInfo			:= ADR(InputArguments),
		cbInputArgInfo			:= SIZEOF(InputArguments),
		pInputArgData			:= ADR(nInputData),
		cbInputArgData			:= nOffset,
		pInputWriteData			:= 0,
		cbInputWriteData		:= 0,
		nNumberOfOutputArguments:= nNumberOfOutputArguments,	(* 3 *)
		pOutputArgInfo			:= ADR(stOutputArgInfo),
		cbOutputArgInfo			:= SIZEOF(stOutputArgInfo),
		pOutputArgInfoAndData	:= ADR(stOutputArgInfoAndData),
		cbOutputArgInfoAndData	:= SIZEOF(stOutputArgInfoAndData),
		Timeout					:= Timeout
	);
	IF NOT fbUA_MethodCall.Busy THEN
		fbUA_MethodCall(Execute := FALSE, cbRead_R => cbReadData_R);

		IF NOT fbUA_MethodCall.Error THEN
			(*  *)
			iReadStateReqState 	:= iReadStateReqState + 1; (* Release handle *)
			nAdsState := stOutputArgInfoAndData.stADSReadState.nAdsState;
			nDeviceState := stOutputArgInfoAndData.stADSReadState.nDeviceState;		
		ELSE
			bError				:= TRUE;
			nErrorID			:= fbUA_MethodCall.ErrorID;
			iReadStateReqState 	:= 3; (* Release handle *)
		END_IF
	END_IF


3:	(* Release Method Handle *)
	fbUA_MethodReleaseHandle(
		Execute			:= TRUE,
		ConnectionHdl	:= nConnectionHdl,
		MethodHdl		:= nMethodHdl,
		Timeout			:= Timeout
	);

	IF NOT fbUA_MethodReleaseHandle.Busy THEN
		fbUA_MethodReleaseHandle(Execute := FALSE);
		bBusy := FALSE;
		IF NOT fbUA_MethodReleaseHandle.Error THEN
			(* session closed *)
			bDone := TRUE;
			iReadStateReqState 	:= 0; (* idle *)
		ELSE
			bError				:= TRUE;
			nErrorID			:= fbUA_MethodReleaseHandle.ErrorID;
			iReadStateReqState 	:= 0; (* idle *)
		END_IF
	END_IF
END_CASE

ACTION M_Init:
bInputDataError := FALSE; 
nOffset := 0;
MEMSET(ADR(InputArguments),0,SIZEOF(InputArguments));
MEMSET(ADR(nInputData),0,SIZEOF(nInputData));

nArg := 1;
(*sNetID := sAmsNetID;*)	(********** NET ID **********)
InputArguments[nArg].DataType			:= eUAType_String;
InputArguments[nArg].ValueRank			:= -1; 						(* Scalar = -1 or Array *)
InputArguments[nArg].ArrayDimensions[1]	:= 0; 						(* Number of Dimension in case its an array *)
InputArguments[nArg].nLenData			:= INT_TO_UDINT(LEN(sNetId)) + 1;			(* Length if its a STRING *)
IF nOffset + INT_TO_UDINT(LEN(sNetId))+1 > nInputArgSize THEN 
	bInputDataError := TRUE;
	RETURN;
ELSE
	MEMCPY(ADR(nInputData)+nOffset,ADR(sNetId),INT_TO_UDINT(LEN(sNetId))+1);				(* VALUE in BYTES FORM *)
	nOffset := nOffset + INT_TO_UDINT(LEN(sNetId))+1;
END_IF

nArg := nArg + 1;
(* nPort := 851;*)			(********** PORT **********)
InputArguments[nArg].DataType			:= eUAType_Int16;
InputArguments[nArg].ValueRank			:= -1; 						(* Scalar = -1 or Array *)
InputArguments[nArg].ArrayDimensions[1]	:= 0; 						(* Number of Dimension in case its an array *)
InputArguments[nArg].nLenData			:= SIZEOF(nPort);			(* Length if its a STRING *)
IF nOffset + SIZEOF(nPort) > nInputArgSize THEN 
	bInputDataError := TRUE;
	RETURN;
ELSE
	MEMCPY(ADR(nInputData)+nOffset,ADR(nPort),SIZEOF(nPort));			(* VALUE in BYTES FORM *)
	nOffset := nOffset + SIZEOF(nPort);
END_IF

//************** Prepare Output Argument information ***********
stOutputArgInfo[1].nLenData := SIZEOF(stOutputArgInfoAndData.stADSReadState.nAdsState);
stOutputArgInfo[2].nLenData := SIZEOF(stOutputArgInfoAndData.stADSReadState.nDeviceState); 
stOutputArgInfo[3].nLenData := 0;
END_ACTION

END_FUNCTION_BLOCK

// ---- POUs/PRG_ADSWriteControlReq.TcPOU
PROGRAM PRG_ADSWriteControlReq
VAR
	fbUA_Connect			: UA_Connect;
	SessionConnectInfo		: ST_UASessionConnectInfo;
	sOpcUA_URL				: STRING(MAX_STRING_LENGTH);
	nConnectionHdl			: DWORD;

	fbUA_GetNamespaceIndex 	: UA_GetNamespaceIndex;
	nNamespaceIndex			: UINT;

	fbUA_NodeReleaseHandle	: UA_NodeReleaseHandle;
	
	fbUA_MethodCall_ADSWriteControlReq	: UA_MethodCall_ADSWriteControlReq;
	
	fbUA_Disconnect		: UA_Disconnect;
		
	bTest		: BOOL:= TRUE;
	bDone		: BOOL;
	bBusy		: BOOL;
	bError		: BOOL;
	nErrorID	: DWORD;
	iState		: INT;
END_VAR

CASE iState OF
0:	(* idle *)
	IF bTest THEN
		bTest	:= FALSE;
		bError	:= FALSE;
		nErrorID	:= 0;

		(* Parameterize *)
		sOpcUA_URL						:= 'opc.tcp://Pujak-nb:4840';	(* OpcUA Url of the device with ip address *)

		SessionConnectInfo.tConnectTimeout 	:= t#1s;
		SessionConnectInfo.tSessionTimeout 	:= t#1s;
		SessionConnectInfo.sApplicationName	:= '';
//		SessionConnectInfo.sApplicationUri 	:= '';
		SessionConnectInfo.eSecurityMode 		:= eUASecurityMsgMode_None;
		SessionConnectInfo.eSecurityPolicyUri 	:= eUASecurityPolicy_None;
		SessionConnectInfo.eTransportProfileUri := eUATransportProfileUri_UATcp;

		iState	:= iState + 1;	(* open ua session *)
	END_IF

1:	(* open UA session *)
	fbUA_Connect(
		Execute				:= TRUE,
		ServerURL			:= sOpcUA_URL,
		SessionConnectInfo	:= SessionConnectInfo,
		Timeout				:= T#5S,
		ConnectionHdl		=> nConnectionHdl
	);

	IF NOT fbUA_Connect.Busy THEN
		fbUA_Connect(Execute := FALSE);

		IF NOT fbUA_Connect.Error THEN
			(* session open *)
			iState := iState + 1;	(* get namespace index *)
		ELSE
			bError			:= TRUE;
			nErrorID		:= fbUA_Connect.ErrorID;
			nConnectionHdl	:= 0;
			iState 			:= 0; (* idle *)
		END_IF
	END_IF


2:	(* GetNS Index *)
	fbUA_GetNamespaceIndex(
		Execute			:= TRUE,
		ConnectionHdl	:= nConnectionHdl,
		NamespaceUri	:= 'ADSAMS',
		NamespaceIndex	=> nNamespaceIndex
	);

	IF NOT fbUA_GetNamespaceIndex.Busy THEN
		fbUA_GetNamespaceIndex(Execute := FALSE);

		IF NOT fbUA_GetNamespaceIndex.Error THEN
			(* session closed *)
			iState 		:= iState + 1; (* method *)
		ELSE
			bError		:= TRUE;
			nErrorID	:= fbUA_GetNamespaceIndex.ErrorID;
			iState 		:= 4; (* close session *)
		END_IF
	END_IF

3:	(*  Method  *)
	fbUA_MethodCall_ADSWriteControlReq(
		bExecute		:= TRUE,
		nConnectionHdl	:= nConnectionHdl,
		nNamespaceIndex	:= nNamespaceIndex,
		sNetID			:= '127.0.0.1.1.1',
		nPort			:= 10000, // TC Restart
		nAdsState		:= 2,
		nDeviceState	:= 0 );
		// nPort := 851, nAdsState := 2, nDeviceState := 0 );
	IF NOT fbUA_MethodCall_ADSWriteControlReq.bBusy THEN
		fbUA_MethodCall_ADSWriteControlReq(	bExecute 	 := FALSE );
		IF NOT fbUA_MethodCall_ADSWriteControlReq.bError THEN
			(* session closed *)
			iState 		:= iState + 1; (* close session *)
		ELSE
			bError		:= TRUE;
			nErrorID	:= fbUA_MethodCall_ADSWriteControlReq.nErrorID;
			iState 		:= 4; (* close session *)
		END_IF
	END_IF


4:	(* close session *)
	fbUA_Disconnect(
		Execute			:= TRUE,
		ConnectionHdl	:= nConnectionHdl
	);

	IF NOT fbUA_Disconnect.Busy THEN
		fbUA_Disconnect(Execute := FALSE);
		bBusy := FALSE; 
		IF NOT fbUA_Disconnect.Error THEN
			(* session closed *)
			iState 		:= 0; (* idle *)
			IF NOT bError THEN 
				bDone 	:= TRUE;
			END_IF
		ELSE
			bError			:= TRUE;
			nErrorID		:= fbUA_Disconnect.ErrorID;
			iState 			:= 0; (* idle *)
			nConnectionHdl	:= 0;
		END_IF
	END_IF
END_CASE

END_PROGRAM

// ---- BECKHOFF SPECIFIC helper library/POUs/MethodCall/UA_MethodCall_ADSWriteControlReq.TcPOU
FUNCTION_BLOCK UA_MethodCall_ADSWriteControlReq
VAR_INPUT
	bExecute			: BOOL;
	nConnectionHdl		: DWORD;
	nNamespaceIndex		: UINT; 		(* to be retrieved using UA_GetNamespaceIndex *)
	sNetID				: T_AmsNetId; 	(* AmsNetId OF the Target *)
	nPort				: INT; 			(* Port number	*)
	nAdsState			: DINT;			(* IndexGroup*)
	nDeviceState		: DINT; 		(* IndexOffset*)
	pWriteData			: PVOID;
	cbWriteData			: UDINT;		(* Count of bytes to be written*)
	Timeout				: TIME := DEFAULT_ADS_TIMEOUT;
END_VAR
VAR_OUTPUT
	bDone				: BOOL;
	bBusy				: BOOL;
	bError				: BOOL;
	nErrorID			: DWORD;
END_VAR
VAR
	iWriteControlReqState	: INT;
	RTrig					: R_TRIG;

	fbUA_MethodGetHandle: UA_MethodGetHandle;
	nMethodHdl			: DWORD;
	ObjectNodeID		: ST_UANodeID;
	MethodNodeID		: ST_UANodeID;

	fbUA_MethodCall		: UA_MethodCall;
	InputArguments		: ARRAY [1..nNumberOfInputArguments] OF ST_UAMethodArgInfo; (*WriteControlReq has 5 input parameters *)
	nNumberOfOutputArguments_R	: UDINT;
	nArg				: INT;
	nInputData			: ARRAY [1..nInputArgSize] OF BYTE;(* NetID(24)+ Port(2)+ ADSState(4)+ DeviceState(4)*)
	nOffset				: UDINT;
	
	fbUA_MethodReleaseHandle: UA_MethodReleaseHandle;
	bInputDataError 		: BOOL; 
END_VAR
VAR CONSTANT
	nInputArgSize			: UDINT := 34; // (* NetID(24)+ Port(2)+ ADSState(4)+ DeviceState(4)*)
	nNumberOfInputArguments : UDINT := 5;
	nNumberOfOutputArguments: UDINT := 0;
END_VAR

(*
ADSWriteControlReq(
******** Input Arguments ********
	string sNetID, 		: AmsNetId of the Target
	int16 Port,			: Port number	
	int32 AdsState,		: Ads State
	int32 DeviceState	: Device State
	ByteString Data		: Data to be written to the device
******** Output Arguments ********
	
);
*)
RTrig(CLK:= bExecute);

CASE iWriteControlReqState OF

0:	(* Get Method Handle *)
	IF RTrig.Q THEN
		bBusy		:= TRUE;
		bDone 		:= FALSE;
		bError		:= FALSE;
		nErrorID	:= 0;
		ObjectNodeID.eIdentifierType 	:= eUAIdentifierType_String;
		ObjectNodeID.nNamespaceIndex 	:= nNamespaceIndex;
		ObjectNodeID.sIdentifier		:= 'ADSAMS';
	
		MethodNodeID.eIdentifierType 	:= eUAIdentifierType_String;
		MethodNodeID.nNamespaceIndex 	:= nNamespaceIndex;
		MethodNodeID.sIdentifier		:= 'ADSAMS.AdsWriteControlReq';

		M_Init();
		IF bInputDataError = FALSE THEN
			iWriteControlReqState 	:= iWriteControlReqState + 1;
		ELSE
			bBusy		:= FALSE;
			bError 		:= TRUE;
			nErrorID 	:= DEVICE_INVALIDSIZE; //16#705 parameter size not correct
		END_IF		
	END_IF


1:	(* Method Get Handle *)
	fbUA_MethodGetHandle(
			Execute			:= TRUE,
			ConnectionHdl	:= nConnectionHdl,
			ObjectNodeID	:= ObjectNodeID,
			MethodNodeID 	:= MethodNodeID,
			Timeout			:= Timeout,
			MethodHdl		=> nMethodHdl
		);
	IF NOT fbUA_MethodGetHandle.Busy THEN
		fbUA_MethodGetHandle(Execute := FALSE);

		IF NOT fbUA_MethodGetHandle.Error THEN
			(*  *)
			iWriteControlReqState := iWriteControlReqState + 1; (* Call Method *)
		ELSE
			bError			:= TRUE;
			nErrorID		:= fbUA_MethodGetHandle.ErrorID;
			iWriteControlReqState 	:= 3; (* Release Handle *)
		END_IF
	END_IF


2:	(* Method Call *)
	fbUA_MethodCall(
		Execute					:= TRUE,
		ConnectionHdl			:= nConnectionHdl,
		MethodHdl				:= nMethodHdl,
		nNumberOfInputArguments := nNumberOfInputArguments,		(* 5 *)
		pInputArgInfo			:= ADR(InputArguments),
		cbInputArgInfo			:= SIZEOF(InputArguments),
		pInputArgData			:= ADR(nInputData),
		cbInputArgData			:= nOffset,
		pInputWriteData			:= pWriteData,
		cbInputWriteData		:= cbWriteData,
		nNumberOfOutputArguments:= nNumberOfOutputArguments,		(* 0 *)
		pOutputArgInfo			:= 0,
		cbOutputArgInfo			:= 0,
		pOutputArgInfoAndData	:= ADR(nNumberOfOutputArguments_R),	//minimum output
		cbOutputArgInfoAndData	:= SIZEOF(nNumberOfOutputArguments_R),	//minimum output
		Timeout					:= Timeout
	);

	IF NOT fbUA_MethodCall.Busy THEN
		fbUA_MethodCall(Execute := FALSE);
		IF NOT fbUA_MethodCall.Error THEN
			(*  *)
			iWriteControlReqState 	:= iWriteControlReqState + 1; (* Release handle *)
			(*MEMSET(ADR(Data),0,nMaxNumberofOutputArgBytes);
			MEMCPY(ADR(Data),ADR(OutputArguments),cbData); *)
		ELSE
			bError					:= TRUE;
			nErrorID				:= fbUA_MethodCall.ErrorID;
			iWriteControlReqState	:= 3; (* Release handle *)
		END_IF
	END_IF


3:	(* Release Method Handle *)
	fbUA_MethodReleaseHandle(
		Execute			:= TRUE,
		ConnectionHdl	:= nConnectionHdl,
		MethodHdl		:= nMethodHdl,
		Timeout			:= Timeout
	);

	IF NOT fbUA_MethodReleaseHandle.Busy THEN
		fbUA_MethodReleaseHandle(Execute := FALSE);
		bBusy := FALSE;
		IF NOT fbUA_MethodReleaseHandle.Error THEN
			(* session closed *)
			bDone := TRUE;
			iWriteControlReqState 	:= 0; (* idle *)
		ELSE
			bError			:= TRUE;
			nErrorID		:= fbUA_MethodReleaseHandle.ErrorID;
			iWriteControlReqState 	:= 0; (* idle *)
		END_IF
	END_IF
END_CASE

ACTION M_Init:
bInputDataError := FALSE; 
nOffset := 0;
MEMSET(ADR(InputArguments),0,SIZEOF(InputArguments));
MEMSET(ADR(nInputData),0,SIZEOF(nInputData));

nArg := 1;
(*sNetID := sAmsNetID;*)	(********** NET ID **********);
InputArguments[nArg].DataType			:= eUAType_String;
InputArguments[nArg].ValueRank			:= -1; 							(* Scalar = -1 or Array *)
InputArguments[nArg].ArrayDimensions[1]	:= 0; 							(* Number of Dimension in case its an array *)
InputArguments[nArg].nLenData			:= INT_TO_UDINT(LEN(sNetId)) + 1;				(* Length if its a STRING *)
IF nOffset + INT_TO_UDINT(LEN(sNetId))+1 > nInputArgSize THEN 
	bInputDataError := TRUE;
	RETURN;
ELSE
	MEMCPY(ADR(nInputData)+nOffset,ADR(sNetId),INT_TO_UDINT(LEN(sNetId))+1);				(* VALUE in BYTES FORM *)
	nOffset := nOffset + INT_TO_UDINT(LEN(sNetId))+1;
END_IF

nArg := nArg + 1;
(* nPort := 851;*)			(********** PORT **********)
InputArguments[nArg].DataType			:= eUAType_Int16;
InputArguments[nArg].ValueRank			:= -1; 							(* Scalar = -1 or Array *)
InputArguments[nArg].ArrayDimensions[1]	:= 0; 							(* Number of Dimension in case its an array *)
InputArguments[nArg].nLenData			:= SIZEOF(nPort);				(* Length if its a STRING *)
IF nOffset + SIZEOF(nPort) > nInputArgSize THEN 
	bInputDataError := TRUE;
	RETURN;
ELSE
	MEMCPY(ADR(nInputData)+nOffset,ADR(nPort),SIZEOF(nPort));			(* VALUE in BYTES FORM *)
	nOffset := nOffset + SIZEOF(nPort);
END_IF

nArg := nArg + 1;
(*nAdsState := ;*)	(********** Ads State **********)
InputArguments[nArg].DataType			:= eUAType_Int32;
InputArguments[nArg].ValueRank			:= -1; 							(* Scalar = -1 or Array *)
InputArguments[nArg].ArrayDimensions[1]	:= 0; 							(* Number of Dimension in case its an array *)
InputArguments[nArg].nLenData			:= SIZEOF(nAdsState);			(* Length if its a STRING *)
IF nOffset + SIZEOF(nAdsState) > nInputArgSize THEN 
	bInputDataError := TRUE;
	RETURN;
ELSE
	MEMCPY(ADR(nInputData)+nOffset,ADR(nAdsState),SIZEOF(nAdsState));		(* VALUE in BYTES FORM *)
	nOffset := nOffset + SIZEOF(nAdsState);
END_IF

nArg := nArg + 1;
(*nDeviceState := ; *)		(********** Device State **********)
InputArguments[nArg].DataType			:= eUAType_Int32;
InputArguments[nArg].ValueRank			:= -1; 							(* Scalar = -1 or Array *)
InputArguments[nArg].ArrayDimensions[1]	:= 0; 							(* Number of Dimension in case its an array *)
InputArguments[nArg].nLenData			:= SIZEOF(nDeviceState);		(* Length if its a STRING *)
IF nOffset + SIZEOF(nDeviceState) > nInputArgSize THEN 
	bInputDataError := TRUE;
	RETURN;
ELSE
	MEMCPY(ADR(nInputData)+nOffset,ADR(nDeviceState),SIZEOF(nDeviceState));	(* VALUE in BYTES FORM *)
	nOffset := nOffset + SIZEOF(nDeviceState);
END_IF

nArg := nArg + 1;
(*Data := ; *)		(*********** WriteData ***********)
InputArguments[nArg].DataType			:= eUAType_ByteString;
InputArguments[nArg].ValueRank			:= -1; 							(* Scalar = -1 or Array *)
InputArguments[nArg].ArrayDimensions[1]	:= 0; 							(* Number of Dimension in case its an array *)
InputArguments[nArg].nLenData			:= cbWriteData;						(* Length if its a STRING *)
END_ACTION

END_FUNCTION_BLOCK

// ---- POUs/PRG_ADSReadWriteReq.TcPOU
PROGRAM PRG_ADSReadWriteReq
VAR
	fbUA_Connect			: UA_Connect;
	SessionConnectInfo		: ST_UASessionConnectInfo;
	sOpcUA_URL				: STRING(MAX_STRING_LENGTH);
	nConnectionHdl			: DWORD;

	fbUA_GetNamespaceIndex 	: UA_GetNamespaceIndex;
	nNamespaceIndex			: UINT;

	fbUA_NodeReleaseHandle	: UA_NodeReleaseHandle;
	
	fbUA_MethodCall_ADSReadWriteReq		: UA_MethodCall_ADSReadWriteReq;
	sHostname		: T_MaxString := 'PujaK-nb';	
	sAddr			: T_IPv4Addr 		:= '';(* String containing an (Ipv4) Internet Protocol dotted address. E.g. '172.16.7.199' *)
	//arrAddr			: T_IPv4AddrArr	:=[ 0, 0, 0, 0];(* Byte array containing an (Ipv4) Internet Protocol dotted address. *)
	//	ReadData		: ARRAY [1..5] OF BYTE;
	stADSReadWriteRes	: ST_ADSReadWriteRes; // T_IPv4AddrArr is to be found here
	stOutputArgInfo		: ST_UAMethodArgInfo;
	fbUA_Disconnect		: UA_Disconnect;
		
	bTest		: BOOL:= TRUE;
	bDone		: BOOL;
	bBusy		: BOOL;
	bError		: BOOL;
	nErrorID	: DWORD;
	iState		: INT;
END_VAR
VAR CONSTANT
	nNumberOfOutputArguments	: UDINT := 1;
END_VAR


CASE iState OF
0:	(* idle *)
	IF bTest THEN
		bTest	:= FALSE;
		bError	:= FALSE;
		nErrorID	:= 0;

		(* Parameterize *)
		sOpcUA_URL								:= 'opc.tcp://Pujak-nb:4840';	(* OpcUA Url of the device with ip address *)

		SessionConnectInfo.tConnectTimeout 		:= T#5S;
		SessionConnectInfo.tSessionTimeout 		:= T#1S;
		SessionConnectInfo.sApplicationName		:= '';
//		SessionConnectInfo.sApplicationUri 		:= '';
		SessionConnectInfo.eSecurityMode 		:= eUASecurityMsgMode_None;
		SessionConnectInfo.eSecurityPolicyUri 	:= eUASecurityPolicy_None;
		SessionConnectInfo.eTransportProfileUri := eUATransportProfileUri_UATcp;

		iState	:= iState + 1;	(* open ua session *)
	END_IF

1:	(* open UA session *)
	fbUA_Connect(
		Execute				:= TRUE,
		ServerURL			:= sOpcUA_URL,
		SessionConnectInfo	:= SessionConnectInfo,
		Timeout				:= T#5S,
		ConnectionHdl		=> nConnectionHdl
	);

	IF NOT fbUA_Connect.Busy THEN
		fbUA_Connect(Execute := FALSE);

		IF NOT fbUA_Connect.Error THEN
			(* session open *)
			iState := iState + 1;	(* get namespace index *)
		ELSE
			bError			:= TRUE;
			nErrorID		:= fbUA_Connect.ErrorID;
			nConnectionHdl	:= 0;
			iState 			:= 0; (* idle *)
		END_IF
	END_IF


2:	(* GetNS Index *)
	fbUA_GetNamespaceIndex(
		Execute			:= TRUE,
		ConnectionHdl	:= nConnectionHdl,
		NamespaceUri	:= 'ADSAMS',
		NamespaceIndex	=> nNamespaceIndex
	);

	IF NOT fbUA_GetNamespaceIndex.Busy THEN
		fbUA_GetNamespaceIndex(Execute := FALSE);

		IF NOT fbUA_GetNamespaceIndex.Error THEN
			(* session closed *)
			iState 		:= iState + 1; (* method *)
		ELSE
			bError		:= TRUE;
			nErrorID	:= fbUA_GetNamespaceIndex.ErrorID;
			iState 		:= 4; (* close session *)
		END_IF
	END_IF

3:	(*  Method  *)
	(*stOutputArgInfo.DataType := eUAType_ByteString;
	stOutputArgInfo.ValueRank := 1; 
	stOutputArgInfo.ArrayDimensions[1] := 4; *)
	stOutputArgInfo.nLenData := 4;//SIZEOF(stADSReadWriteRes.arrAddr);
	fbUA_MethodCall_ADSReadWriteReq(
		bExecute				:= TRUE,
		nConnectionHdl			:= nConnectionHdl,
		nNamespaceIndex			:= nNamespaceIndex,
		sNetID					:= sPujaNetID, //'127.0.0.1.1.1',
		nPort					:= UINT_TO_INT(AMSPORT_R3_SYSSERV),
		nIndexGroup				:= UDINT_TO_DINT(SYSTEMSERVICE_IPHELPERAPI), // 701
		nIndexOffset			:= UDINT_TO_DINT(IPHELPERAPI_IPADDRBYHOSTNAME), //4
		pWriteData 				:= ADR(sHostname),
		cbWriteData				:= INT_TO_UDINT( LEN( sHostName ) + 1),
		pReadArgInfoAndData		:= ADR(stADSReadWriteRes),
		cbReadArgInfoAndData	:= SIZEOF(stADSReadWriteRes),
		nNumberOfOutputArguments:= nNumberOfOutputArguments,
		pOutputArgInfo			:= ADR(stOutputArgInfo),
		cbOutputArgInfo			:= SIZEOF(stOutputArgInfo)		
		);

	IF NOT fbUA_MethodCall_ADSReadWriteReq.bBusy THEN
		fbUA_MethodCall_ADSReadWriteReq(bExecute := FALSE);
		IF NOT fbUA_MethodCall_ADSReadWriteReq.bError THEN
			(* session closed *)
			iState 		:= iState + 1; (* close session *)
			sAddr		:= F_CreateIPv4Addr( stADSReadWriteRes.arrAddr );
		ELSE
			bError		:= TRUE;
			nErrorID	:= fbUA_MethodCall_ADSReadWriteReq.nErrorID;
			iState 		:= 4; (* close session *)
		END_IF
	END_IF


4:	(* close session *)
	fbUA_Disconnect(
		Execute			:= TRUE,
		ConnectionHdl	:= nConnectionHdl
	);

	IF NOT fbUA_Disconnect.Busy THEN
		fbUA_Disconnect(Execute := FALSE);
		bBusy := FALSE;
		IF NOT fbUA_Disconnect.Error THEN
			(* session closed *)
			iState 		:= 0; (* idle *)
			IF NOT bError THEN 
				bDone 	:= TRUE;
			END_IF
		ELSE
			bError			:= TRUE;
			nErrorID		:= fbUA_Disconnect.ErrorID;
			iState 			:= 0; (* idle *)
			nConnectionHdl	:= 0;
		END_IF
	END_IF
END_CASE

END_PROGRAM

